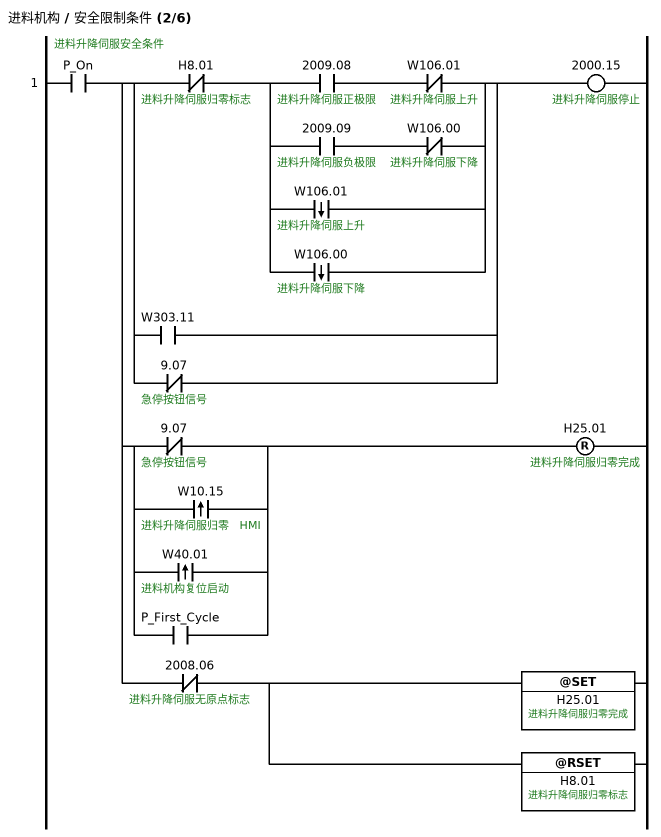
; [picture p72: 进料机构 / 安全限制条件, rungs 1-1]
; rung 1: 进料升降伺服安全条件
LD P_On
OUT TR0
LDNOT H8.01  ; 进料升降伺服归零标志
LD 2009.08  ; 进料升降伺服正极限
ANDNOT W106.01  ; 进料升降伺服上升
LD 2009.09  ; 进料升降伺服负极限
ANDNOT W106.00  ; 进料升降伺服下降
ORLD
%OR W106.01  ; 进料升降伺服上升
%OR W106.00  ; 进料升降伺服下降
ANDLD
OR W303.11
ORNOT 9.07  ; 急停按钮信号
ANDLD
OUT 2000.15  ; 进料升降伺服停止
LD TR0
LDNOT 9.07  ; 急停按钮信号
@OR W10.15  ; 进料升降伺服归零   HMI
@OR W40.01  ; 进料机构复位启动
OR P_First_Cycle
ANDLD
RSET H25.01  ; 进料升降伺服归零完成
LD TR0
ANDNOT 2008.06  ; 进料升降伺服无原点标志
@SET H25.01  ; 进料升降伺服归零完成
@RSET H8.01  ; 进料升降伺服归零标志

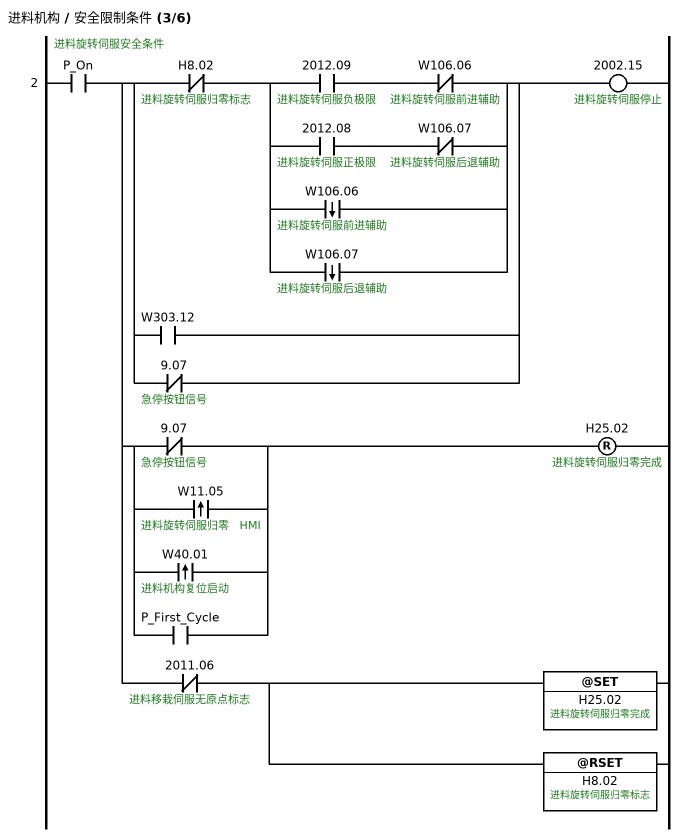
; rung 2: 进料旋转伺服安全条件
LD P_On
OUT TR0
LDNOT H8.02  ; 进料旋转伺服归零标志
LD 2012.09  ; 进料旋转伺服负极限
ANDNOT W106.06  ; 进料旋转伺服前进辅助
LD 2012.08  ; 进料旋转伺服正极限
ANDNOT W106.07  ; 进料旋转伺服后退辅助
ORLD
%OR W106.06  ; 进料旋转伺服前进辅助
%OR W106.07  ; 进料旋转伺服后退辅助
ANDLD
OR W303.12
ORNOT 9.07  ; 急停按钮信号
ANDLD
OUT 2002.15  ; 进料旋转伺服停止
LD TR0
LDNOT 9.07  ; 急停按钮信号
@OR W11.05  ; 进料旋转伺服归零   HMI
@OR W40.01  ; 进料机构复位启动
OR P_First_Cycle
ANDLD
RSET H25.02  ; 进料旋转伺服归零完成
LD TR0
ANDNOT 2011.06  ; 进料移栽伺服无原点标志
@SET H25.02  ; 进料旋转伺服归零完成
@RSET H8.02  ; 进料旋转伺服归零标志

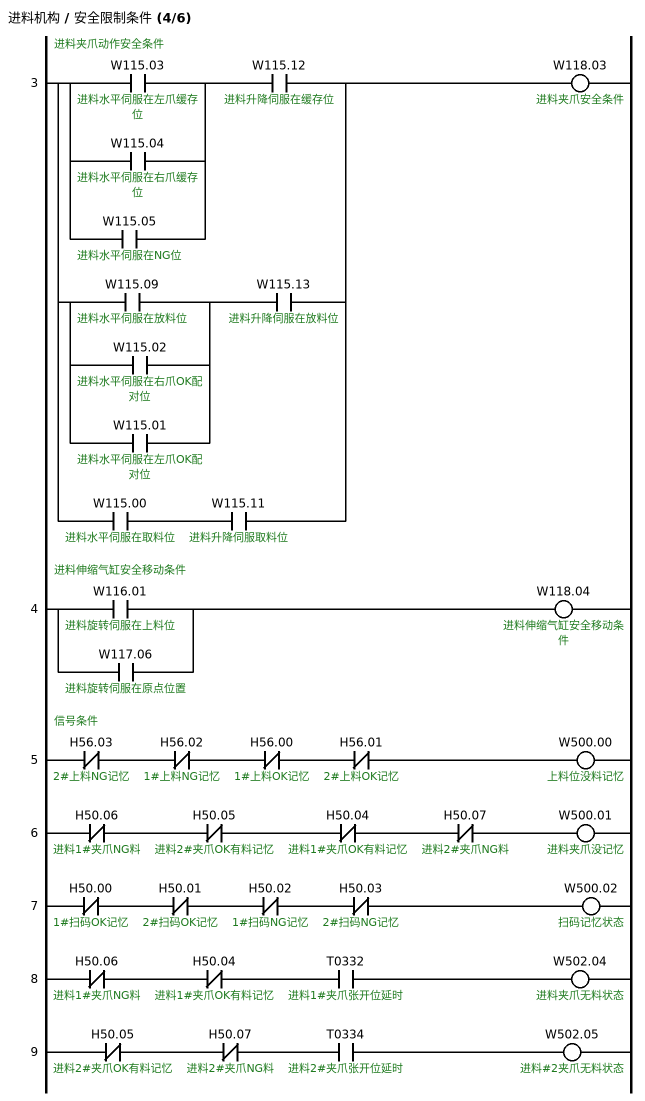
; rung 3: 进料夹爪动作安全条件
LD W115.03  ; 进料水平伺服在左爪缓存位
OR W115.04  ; 进料水平伺服在右爪缓存位
OR W115.05  ; 进料水平伺服在NG位
AND W115.12  ; 进料升降伺服在缓存位
LD W115.09  ; 进料水平伺服在放料位
OR W115.02  ; 进料水平伺服在右爪OK配对位
OR W115.01  ; 进料水平伺服在左爪OK配对位
AND W115.13  ; 进料升降伺服在放料位
ORLD
LD W115.00  ; 进料水平伺服在取料位
AND W115.11  ; 进料升降伺服取料位
ORLD
OUT W118.03  ; 进料夹爪安全条件
; rung 4: 进料伸缩气缸安全移动条件
LD W116.01  ; 进料旋转伺服在上料位
OR W117.06  ; 进料旋转伺服在原点位置
OUT W118.04  ; 进料伸缩气缸安全移动条件
; rung 5: 信号条件
LDNOT H56.03  ; 2#上料NG记忆
ANDNOT H56.02  ; 1#上料NG记忆
ANDNOT H56.00  ; 1#上料OK记忆
ANDNOT H56.01  ; 2#上料OK记忆
OUT W500.00  ; 上料位没料记忆
; rung 6
LDNOT H50.06  ; 进料1#夹爪NG料
ANDNOT H50.05  ; 进料2#夹爪OK有料记忆
ANDNOT H50.04  ; 进料1#夹爪OK有料记忆
ANDNOT H50.07  ; 进料2#夹爪NG料
OUT W500.01  ; 进料夹爪没记忆
; rung 7
LDNOT H50.00  ; 1#扫码OK记忆
ANDNOT H50.01  ; 2#扫码OK记忆
ANDNOT H50.02  ; 1#扫码NG记忆
ANDNOT H50.03  ; 2#扫码NG记忆
OUT W500.02  ; 扫码记忆状态
; rung 8
LDNOT H50.06  ; 进料1#夹爪NG料
ANDNOT H50.04  ; 进料1#夹爪OK有料记忆
AND T0332  ; 进料1#夹爪张开位延时
OUT W502.04  ; 进料夹爪无料状态
; rung 9
LDNOT H50.05  ; 进料2#夹爪OK有料记忆
ANDNOT H50.07  ; 进料2#夹爪NG料
AND T0334  ; 进料2#夹爪张开位延时
OUT W502.05  ; 进料#2夹爪无料状态

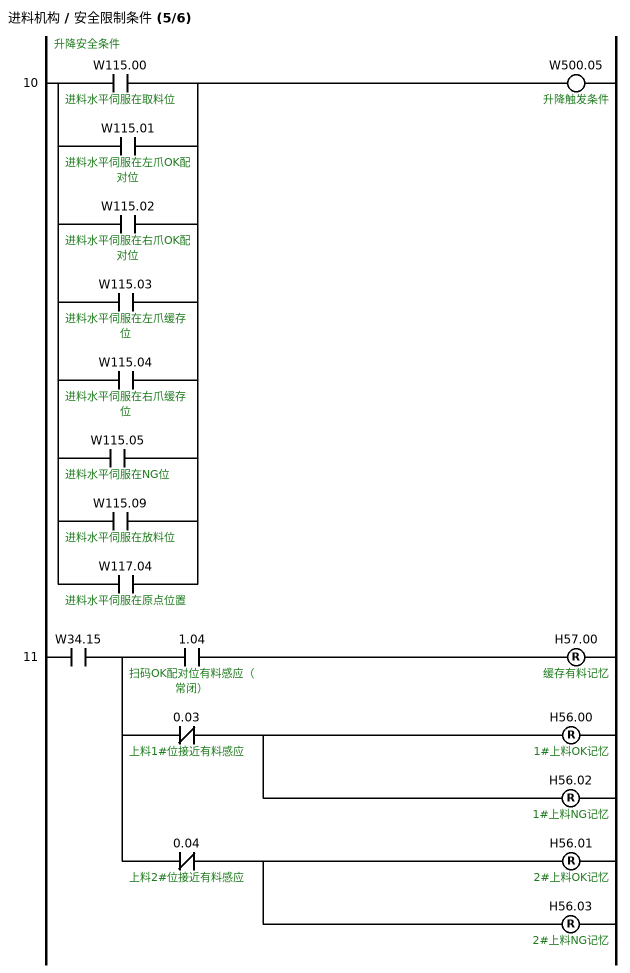
; rung 10: 升降安全条件
LD W115.00  ; 进料水平伺服在取料位
OR W115.01  ; 进料水平伺服在左爪OK配对位
OR W115.02  ; 进料水平伺服在右爪OK配对位
OR W115.03  ; 进料水平伺服在左爪缓存位
OR W115.04  ; 进料水平伺服在右爪缓存位
OR W115.05  ; 进料水平伺服在NG位
OR W115.09  ; 进料水平伺服在放料位
OR W117.04  ; 进料水平伺服在原点位置
OUT W500.05  ; 升降触发条件
; rung 11
LD W34.15
OUT TR0
AND 1.04  ; 扫码OK配对位有料感应（常闭）
RSET H57.00  ; 缓存有料记忆
LD TR0
ANDNOT 0.03  ; 上料1#位接近有料感应
RSET H56.00  ; 1#上料OK记忆
RSET H56.02  ; 1#上料NG记忆
LD TR0
ANDNOT 0.04  ; 上料2#位接近有料感应
RSET H56.01  ; 2#上料OK记忆
RSET H56.03  ; 2#上料NG记忆

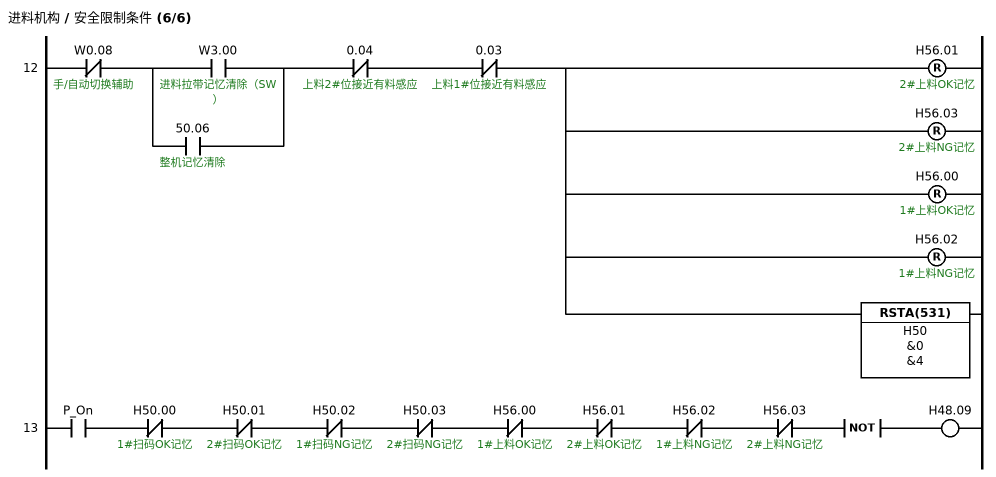
; rung 12
LDNOT W0.08  ; 手/自动切换辅助
LD W3.00  ; 进料拉带记忆清除（SW）
OR 50.06  ; 整机记忆清除
ANDLD
ANDNOT 0.04  ; 上料2#位接近有料感应
ANDNOT 0.03  ; 上料1#位接近有料感应
RSET H56.01  ; 2#上料OK记忆
RSET H56.03  ; 2#上料NG记忆
RSET H56.00  ; 1#上料OK记忆
RSET H56.02  ; 1#上料NG记忆
RSTA(531) H50 &0 &4
; rung 13
LD P_On
ANDNOT H50.00  ; 1#扫码OK记忆
ANDNOT H50.01  ; 2#扫码OK记忆
ANDNOT H50.02  ; 1#扫码NG记忆
ANDNOT H50.03  ; 2#扫码NG记忆
ANDNOT H56.00  ; 1#上料OK记忆
ANDNOT H56.01  ; 2#上料OK记忆
ANDNOT H56.02  ; 1#上料NG记忆
ANDNOT H56.03  ; 2#上料NG记忆
NOT(520)
OUT H48.09

### Section 扫码自动

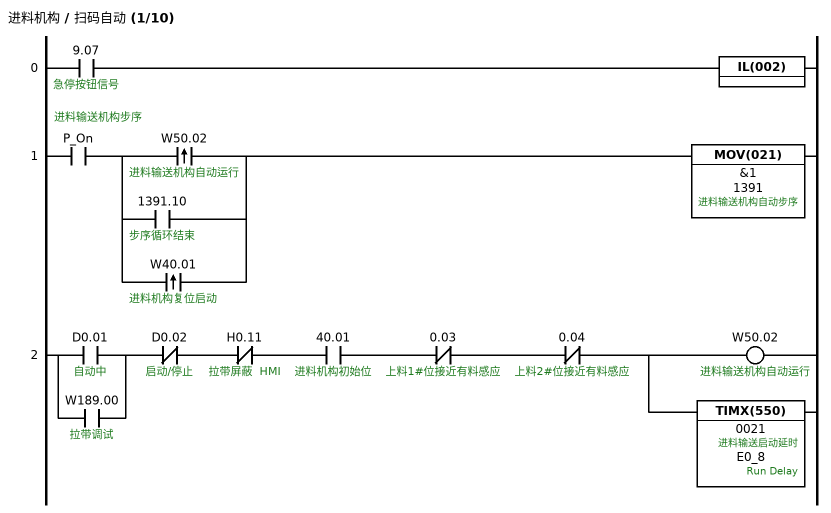
; rung 0
LD 9.07  ; 急停按钮信号
IL(002)
; rung 1: 进料输送机构步序
LD P_On
@LD W50.02  ; 进料输送机构自动运行
OR 1391.10  ; 步序循环结束
@OR W40.01  ; 进料机构复位启动
ANDLD
MOV(021) &1 1391  ; 进料输送机构自动步序
; rung 2
LD D0.01  ; 自动中
OR W189.00  ; 拉带调试
ANDNOT D0.02  ; 启动/停止
ANDNOT H0.11  ; 拉带屏蔽  HMI
AND 40.01  ; 进料机构初始位
ANDNOT 0.03  ; 上料1#位接近有料感应
ANDNOT 0.04  ; 上料2#位接近有料感应
OUT W50.02  ; 进料输送机构自动运行
TIMX(550) 0021 E0_8  ; Run Delay, 进料输送启动延时

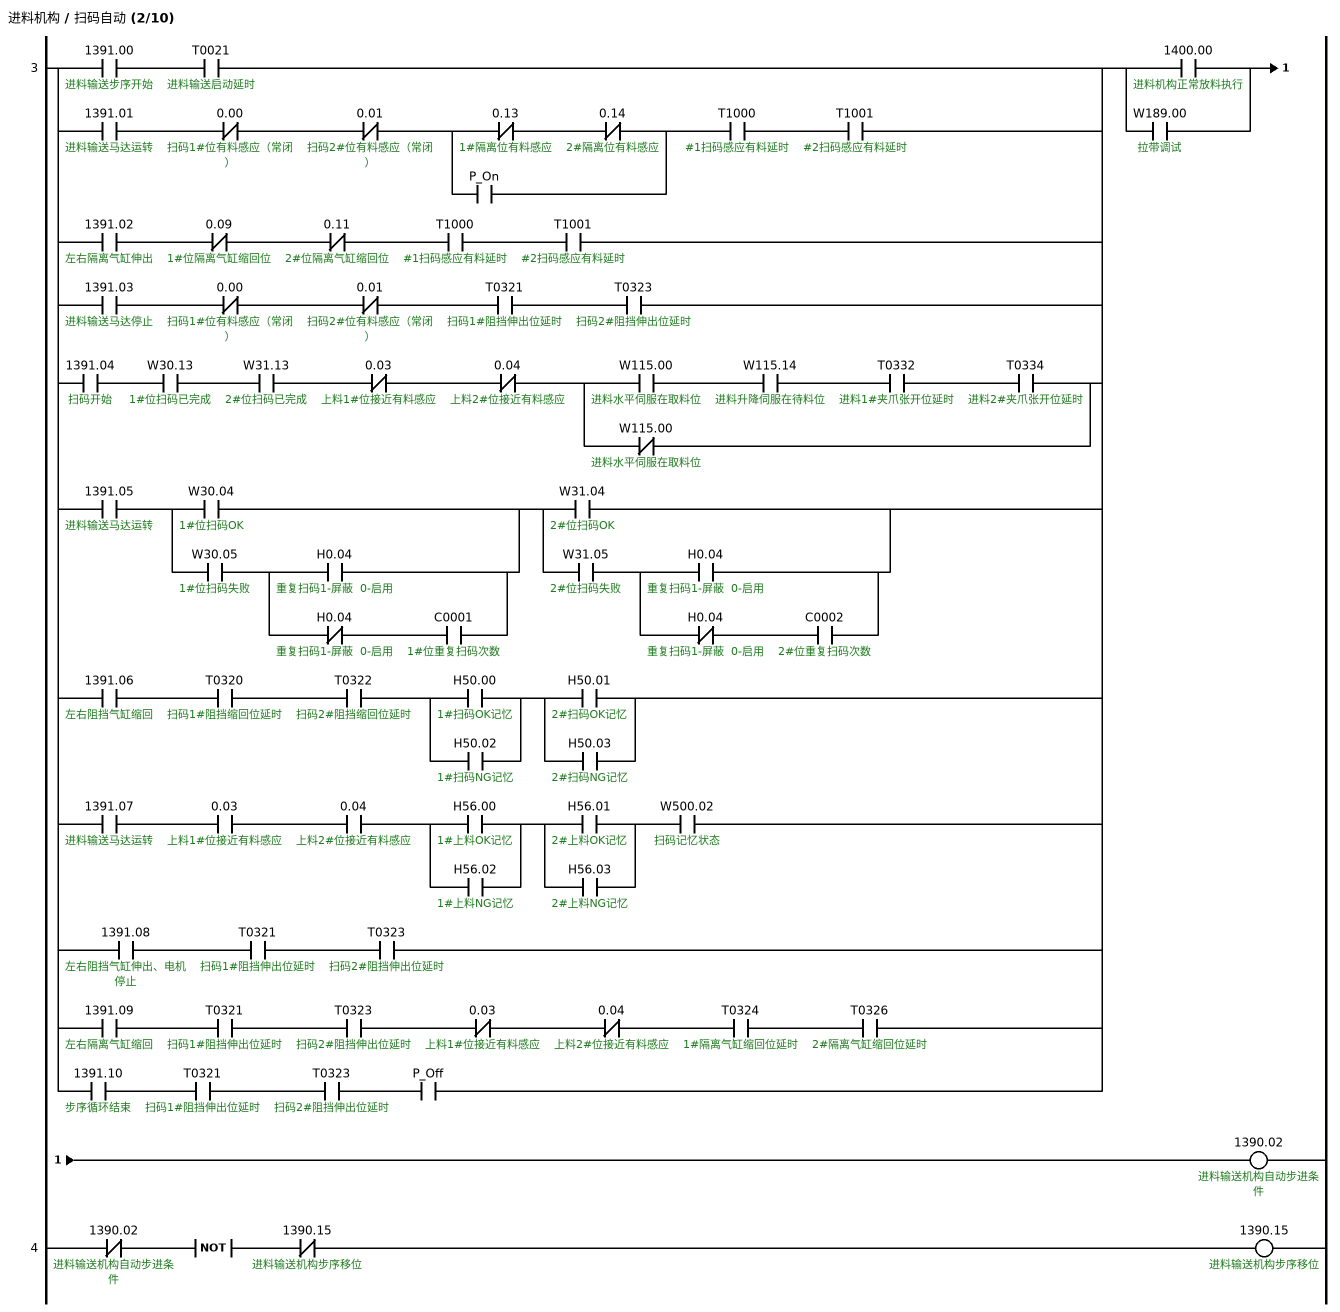
; rung 3
LD 1391.00  ; 进料输送步序开始
AND T0021  ; 进料输送启动延时
LD 1391.01  ; 进料输送马达运转
ANDNOT 0.00  ; 扫码1#位有料感应（常闭）
ANDNOT 0.01  ; 扫码2#位有料感应（常闭）
LDNOT 0.13  ; 1#隔离位有料感应
ANDNOT 0.14  ; 2#隔离位有料感应
OR P_On
ANDLD
AND T1000  ; #1扫码感应有料延时
AND T1001  ; #2扫码感应有料延时
ORLD
LD 1391.02  ; 左右隔离气缸伸出
ANDNOT 0.09  ; 1#位隔离气缸缩回位
ANDNOT 0.11  ; 2#位隔离气缸缩回位
AND T1000  ; #1扫码感应有料延时
AND T1001  ; #2扫码感应有料延时
ORLD
LD 1391.03  ; 进料输送马达停止
ANDNOT 0.00  ; 扫码1#位有料感应（常闭）
ANDNOT 0.01  ; 扫码2#位有料感应（常闭）
AND T0321  ; 扫码1#阻挡伸出位延时
AND T0323  ; 扫码2#阻挡伸出位延时
ORLD
LD 1391.04  ; 扫码开始
AND W30.13  ; 1#位扫码已完成
AND W31.13  ; 2#位扫码已完成
ANDNOT 0.03  ; 上料1#位接近有料感应
ANDNOT 0.04  ; 上料2#位接近有料感应
LD W115.00  ; 进料水平伺服在取料位
AND W115.14  ; 进料升降伺服在待料位
AND T0332  ; 进料1#夹爪张开位延时
AND T0334  ; 进料2#夹爪张开位延时
ORNOT W115.00  ; 进料水平伺服在取料位
ANDLD
ORLD
LD 1391.05  ; 进料输送马达运转
LD W30.04  ; 1#位扫码OK
LD W30.05  ; 1#位扫码失败
LD H0.04  ; 重复扫码1-屏蔽  0-启用
LDNOT H0.04  ; 重复扫码1-屏蔽  0-启用
AND C0001  ; 1#位重复扫码次数
ORLD
ANDLD
ORLD
ANDLD
LD W31.04  ; 2#位扫码OK
LD W31.05  ; 2#位扫码失败
LD H0.04  ; 重复扫码1-屏蔽  0-启用
LDNOT H0.04  ; 重复扫码1-屏蔽  0-启用
AND C0002  ; 2#位重复扫码次数
ORLD
ANDLD
ORLD
ANDLD
ORLD
LD 1391.06  ; 左右阻挡气缸缩回
AND T0320  ; 扫码1#阻挡缩回位延时
AND T0322  ; 扫码2#阻挡缩回位延时
LD H50.00  ; 1#扫码OK记忆
OR H50.02  ; 1#扫码NG记忆
ANDLD
LD H50.01  ; 2#扫码OK记忆
OR H50.03  ; 2#扫码NG记忆
ANDLD
ORLD
LD 1391.07  ; 进料输送马达运转
AND 0.03  ; 上料1#位接近有料感应
AND 0.04  ; 上料2#位接近有料感应
LD H56.00  ; 1#上料OK记忆
OR H56.02  ; 1#上料NG记忆
ANDLD
LD H56.01  ; 2#上料OK记忆
OR H56.03  ; 2#上料NG记忆
ANDLD
AND W500.02  ; 扫码记忆状态
ORLD
LD 1391.08  ; 左右阻挡气缸伸出、电机停止
AND T0321  ; 扫码1#阻挡伸出位延时
AND T0323  ; 扫码2#阻挡伸出位延时
ORLD
LD 1391.09  ; 左右隔离气缸缩回
AND T0321  ; 扫码1#阻挡伸出位延时
AND T0323  ; 扫码2#阻挡伸出位延时
ANDNOT 0.03  ; 上料1#位接近有料感应
ANDNOT 0.04  ; 上料2#位接近有料感应
AND T0324  ; 1#隔离气缸缩回位延时
AND T0326  ; 2#隔离气缸缩回位延时
ORLD
LD 1391.10  ; 步序循环结束
AND T0321  ; 扫码1#阻挡伸出位延时
AND T0323  ; 扫码2#阻挡伸出位延时
AND P_Off
ORLD
LD 1400.00  ; 进料机构正常放料执行
OR W189.00  ; 拉带调试
ANDLD
OUT 1390.02  ; 进料输送机构自动步进条件
; rung 4
LDNOT 1390.02  ; 进料输送机构自动步进条件
NOT(520)
ANDNOT 1390.15  ; 进料输送机构步序移位
OUT 1390.15  ; 进料输送机构步序移位

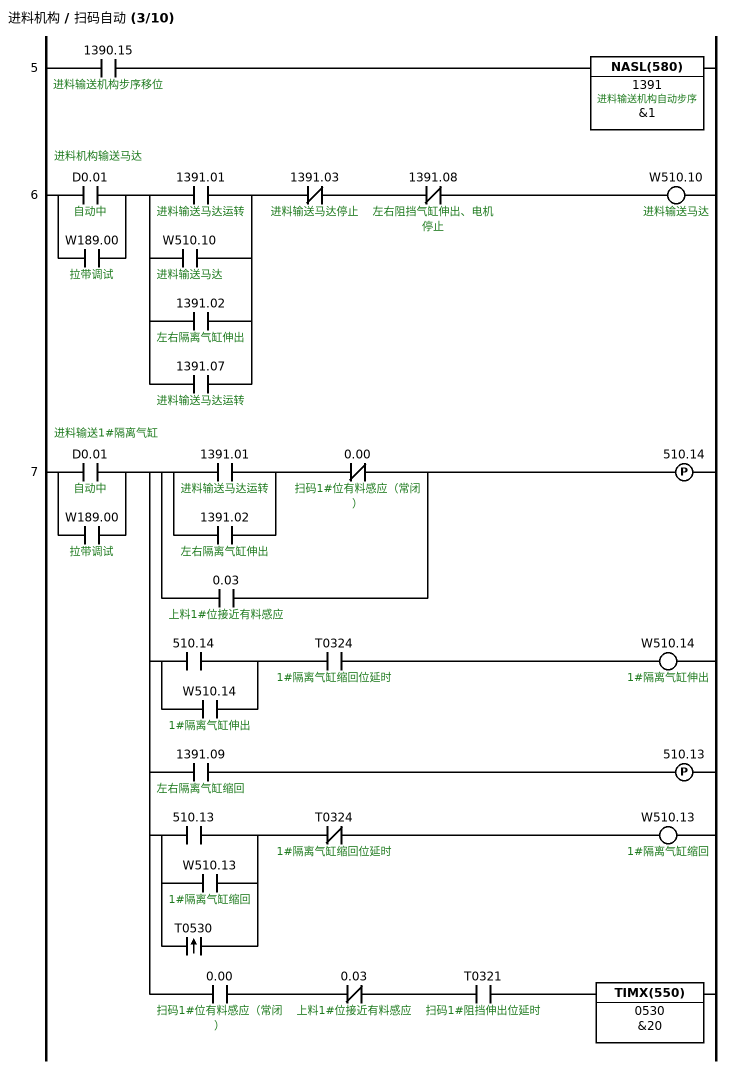
; rung 5
LD 1390.15  ; 进料输送机构步序移位
NASL(580) 1391 &1  ; 进料输送机构自动步序
; rung 6: 进料机构输送马达
LD D0.01  ; 自动中
OR W189.00  ; 拉带调试
LD 1391.01  ; 进料输送马达运转
OR W510.10  ; 进料输送马达
OR 1391.02  ; 左右隔离气缸伸出
OR 1391.07  ; 进料输送马达运转
ANDLD
ANDNOT 1391.03  ; 进料输送马达停止
ANDNOT 1391.08  ; 左右阻挡气缸伸出、电机停止
OUT W510.10  ; 进料输送马达
; rung 7: 进料输送1#隔离气缸
LD D0.01  ; 自动中
OR W189.00  ; 拉带调试
OUT TR0
LD 1391.01  ; 进料输送马达运转
OR 1391.02  ; 左右隔离气缸伸出
ANDNOT 0.00  ; 扫码1#位有料感应（常闭）
OR 0.03  ; 上料1#位接近有料感应
ANDLD
DIFU(013) 510.14
LD TR0
LD 510.14
OR W510.14  ; 1#隔离气缸伸出
ANDLD
AND T0324  ; 1#隔离气缸缩回位延时
OUT W510.14  ; 1#隔离气缸伸出
LD TR0
AND 1391.09  ; 左右隔离气缸缩回
DIFU(013) 510.13
LD TR0
LD 510.13
OR W510.13  ; 1#隔离气缸缩回
@OR T0530
ANDLD
ANDNOT T0324  ; 1#隔离气缸缩回位延时
OUT W510.13  ; 1#隔离气缸缩回
LD TR0
AND 0.00  ; 扫码1#位有料感应（常闭）
ANDNOT 0.03  ; 上料1#位接近有料感应
AND T0321  ; 扫码1#阻挡伸出位延时
TIMX(550) 0530 &20

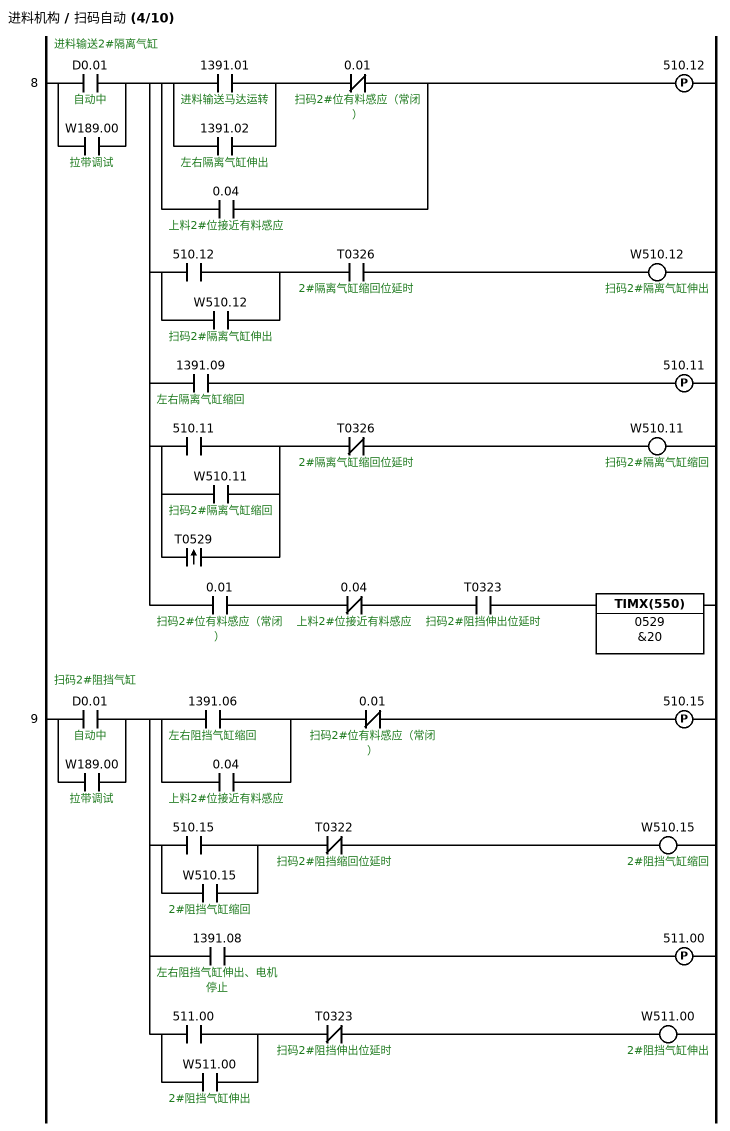
; rung 8: 进料输送2#隔离气缸
LD D0.01  ; 自动中
OR W189.00  ; 拉带调试
OUT TR0
LD 1391.01  ; 进料输送马达运转
OR 1391.02  ; 左右隔离气缸伸出
ANDNOT 0.01  ; 扫码2#位有料感应（常闭）
OR 0.04  ; 上料2#位接近有料感应
ANDLD
DIFU(013) 510.12
LD TR0
LD 510.12
OR W510.12  ; 扫码2#隔离气缸伸出
ANDLD
AND T0326  ; 2#隔离气缸缩回位延时
OUT W510.12  ; 扫码2#隔离气缸伸出
LD TR0
AND 1391.09  ; 左右隔离气缸缩回
DIFU(013) 510.11
LD TR0
LD 510.11
OR W510.11  ; 扫码2#隔离气缸缩回
@OR T0529
ANDLD
ANDNOT T0326  ; 2#隔离气缸缩回位延时
OUT W510.11  ; 扫码2#隔离气缸缩回
LD TR0
AND 0.01  ; 扫码2#位有料感应（常闭）
ANDNOT 0.04  ; 上料2#位接近有料感应
AND T0323  ; 扫码2#阻挡伸出位延时
TIMX(550) 0529 &20
; rung 9: 扫码2#阻挡气缸
LD D0.01  ; 自动中
OR W189.00  ; 拉带调试
OUT TR0
LD 1391.06  ; 左右阻挡气缸缩回
OR 0.04  ; 上料2#位接近有料感应
ANDLD
ANDNOT 0.01  ; 扫码2#位有料感应（常闭）
DIFU(013) 510.15
LD TR0
LD 510.15
OR W510.15  ; 2#阻挡气缸缩回
ANDLD
ANDNOT T0322  ; 扫码2#阻挡缩回位延时
OUT W510.15  ; 2#阻挡气缸缩回
LD TR0
AND 1391.08  ; 左右阻挡气缸伸出、电机停止
DIFU(013) 511.00
LD TR0
LD 511.00
OR W511.00  ; 2#阻挡气缸伸出
ANDLD
ANDNOT T0323  ; 扫码2#阻挡伸出位延时
OUT W511.00  ; 2#阻挡气缸伸出

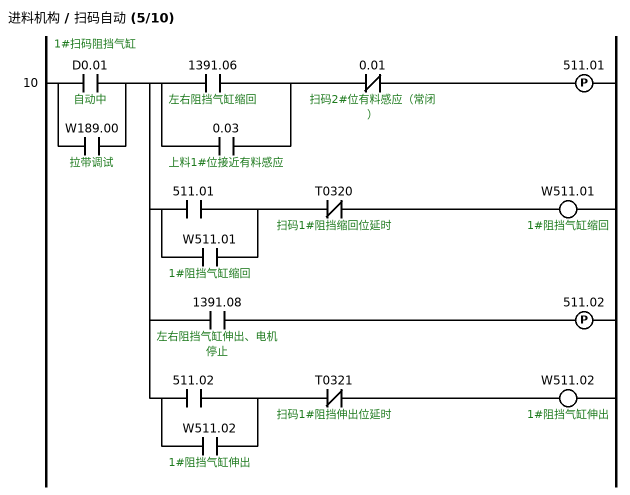
; rung 10: 1#扫码阻挡气缸
LD D0.01  ; 自动中
OR W189.00  ; 拉带调试
OUT TR0
LD 1391.06  ; 左右阻挡气缸缩回
OR 0.03  ; 上料1#位接近有料感应
ANDLD
ANDNOT 0.01  ; 扫码2#位有料感应（常闭）
DIFU(013) 511.01
LD TR0
LD 511.01
OR W511.01  ; 1#阻挡气缸缩回
ANDLD
ANDNOT T0320  ; 扫码1#阻挡缩回位延时
OUT W511.01  ; 1#阻挡气缸缩回
LD TR0
AND 1391.08  ; 左右阻挡气缸伸出、电机停止
DIFU(013) 511.02
LD TR0
LD 511.02
OR W511.02  ; 1#阻挡气缸伸出
ANDLD
ANDNOT T0321  ; 扫码1#阻挡伸出位延时
OUT W511.02  ; 1#阻挡气缸伸出

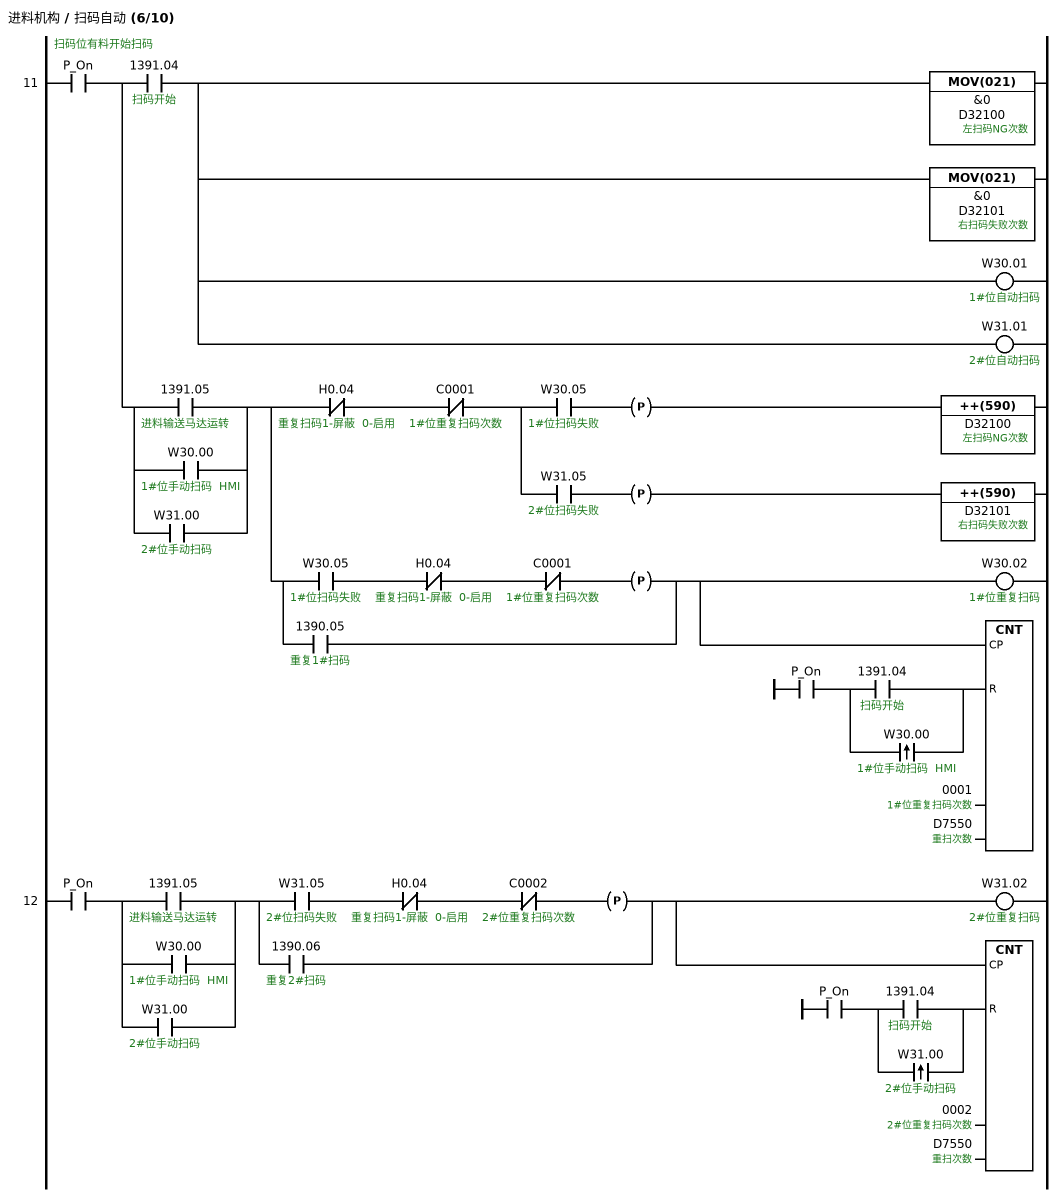
; rung 11: 扫码位有料开始扫码
LD P_On
OUT TR0
AND 1391.04  ; 扫码开始
MOV(021) &0 D32100  ; 左扫码NG次数
MOV(021) &0 D32101  ; 右扫码失败次数
OUT W30.01  ; 1#位自动扫码
OUT W31.01  ; 2#位自动扫码
LD TR0
LD 1391.05  ; 进料输送马达运转
OR W30.00  ; 1#位手动扫码  HMI
OR W31.00  ; 2#位手动扫码
ANDLD
OUT TR0
ANDNOT H0.04  ; 重复扫码1-屏蔽  0-启用
ANDNOT C0001  ; 1#位重复扫码次数
OUT TR1
AND W30.05  ; 1#位扫码失败
UP(521)
++(590) D32100  ; 左扫码NG次数
LD TR1
AND W31.05  ; 2#位扫码失败
UP(521)
++(590) D32101  ; 右扫码失败次数
LD TR0
LD W30.05  ; 1#位扫码失败
ANDNOT H0.04  ; 重复扫码1-屏蔽  0-启用
ANDNOT C0001  ; 1#位重复扫码次数
UP(521)
OR 1390.05  ; 重复1#扫码
ANDLD
OUT W30.02  ; 1#位重复扫码
LD P_On
LD 1391.04  ; 扫码开始
@OR W30.00  ; 1#位手动扫码  HMI
ANDLD
CNT 0001 D7550  ; 重扫次数, 1#位重复扫码次数
; rung 12
LD P_On
LD 1391.05  ; 进料输送马达运转
OR W30.00  ; 1#位手动扫码  HMI
OR W31.00  ; 2#位手动扫码
ANDLD
LD W31.05  ; 2#位扫码失败
ANDNOT H0.04  ; 重复扫码1-屏蔽  0-启用
ANDNOT C0002  ; 2#位重复扫码次数
UP(521)
OR 1390.06  ; 重复2#扫码
ANDLD
OUT W31.02  ; 2#位重复扫码
LD P_On
LD 1391.04  ; 扫码开始
@OR W31.00  ; 2#位手动扫码
ANDLD
CNT 0002 D7550  ; 重扫次数, 2#位重复扫码次数

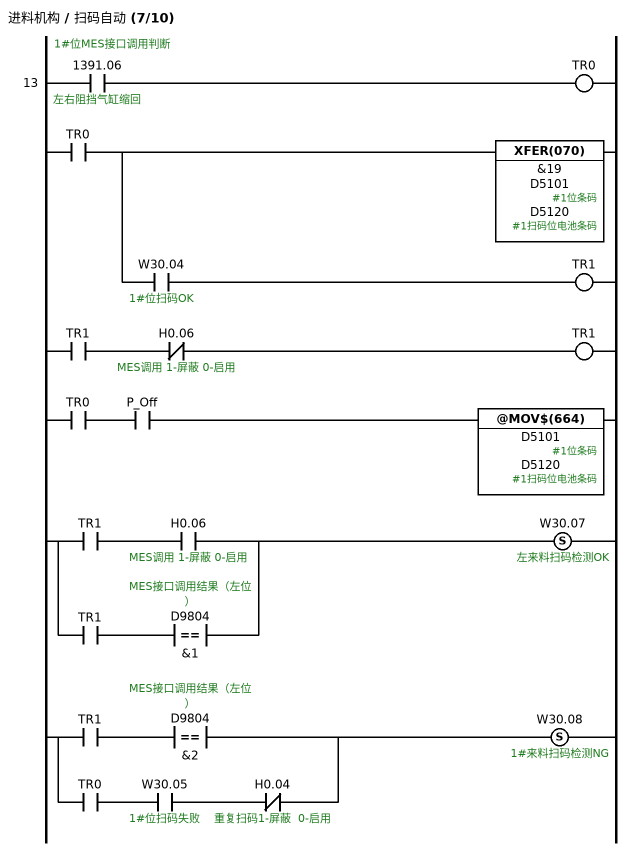
; rung 13: 1#位MES接口调用判断
LD 1391.06  ; 左右阻挡气缸缩回
OUT TR0
AND P_Off
@MOV$(664) D5101 D5120  ; #1位条码, #1扫码位电池条码
LD TR0
XFER(070) &19 D5101 D5120  ; #1位条码, #1扫码位电池条码
AND W30.04  ; 1#位扫码OK
OUT TR1
AND H0.06  ; MES调用 1-屏蔽 0-启用
LD TR1
ANDNOT H0.06  ; MES调用 1-屏蔽 0-启用
OUT TR1
AND=(300) D9804 &1  ; MES接口调用结果（左位）
ORLD
SET W30.07  ; 左来料扫码检测OK
LD TR1
AND=(300) D9804 &2  ; MES接口调用结果（左位）
LD TR0
AND W30.05  ; 1#位扫码失败
ANDNOT H0.04  ; 重复扫码1-屏蔽  0-启用
ORLD
SET W30.08  ; 1#来料扫码检测NG

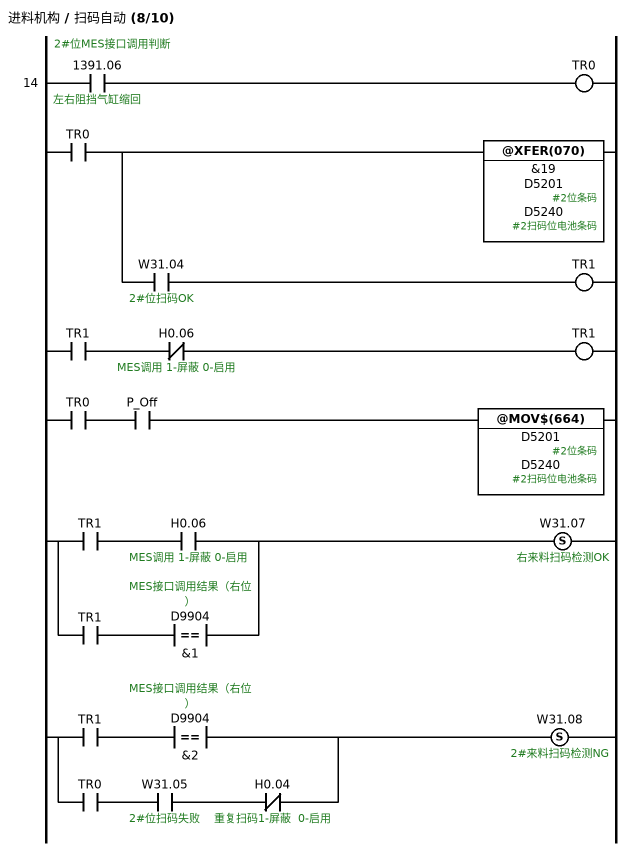
; rung 14: 2#位MES接口调用判断
LD 1391.06  ; 左右阻挡气缸缩回
OUT TR0
AND P_Off
@MOV$(664) D5201 D5240  ; #2位条码, #2扫码位电池条码
LD TR0
@XFER(070) &19 D5201 D5240  ; #2位条码, #2扫码位电池条码
AND W31.04  ; 2#位扫码OK
OUT TR1
AND H0.06  ; MES调用 1-屏蔽 0-启用
LD TR1
ANDNOT H0.06  ; MES调用 1-屏蔽 0-启用
OUT TR1
AND=(300) D9904 &1  ; MES接口调用结果（右位）
ORLD
SET W31.07  ; 右来料扫码检测OK
LD TR1
AND=(300) D9904 &2  ; MES接口调用结果（右位）
LD TR0
AND W31.05  ; 2#位扫码失败
ANDNOT H0.04  ; 重复扫码1-屏蔽  0-启用
ORLD
SET W31.08  ; 2#来料扫码检测NG

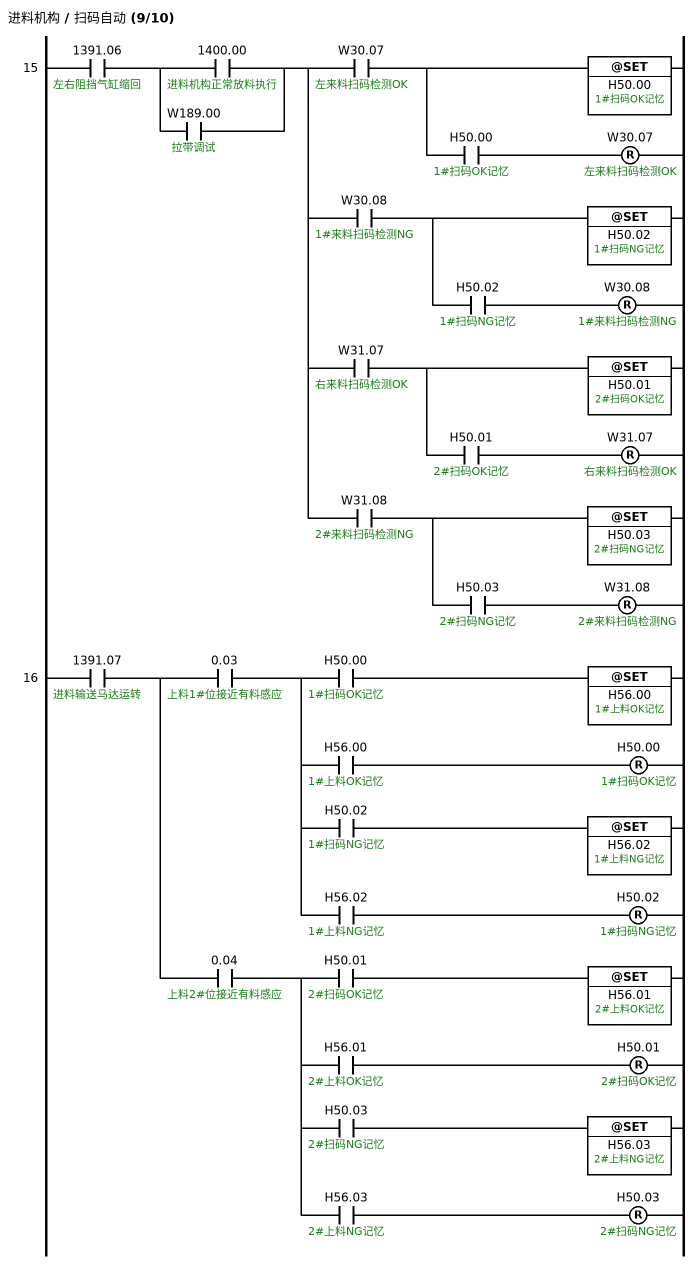
; rung 15
LD 1391.06  ; 左右阻挡气缸缩回
LD 1400.00  ; 进料机构正常放料执行
OR W189.00  ; 拉带调试
ANDLD
OUT TR0
AND W30.07  ; 左来料扫码检测OK
@SET H50.00  ; 1#扫码OK记忆
AND H50.00  ; 1#扫码OK记忆
RSET W30.07  ; 左来料扫码检测OK
LD TR0
AND W30.08  ; 1#来料扫码检测NG
@SET H50.02  ; 1#扫码NG记忆
AND H50.02  ; 1#扫码NG记忆
RSET W30.08  ; 1#来料扫码检测NG
LD TR0
AND W31.07  ; 右来料扫码检测OK
@SET H50.01  ; 2#扫码OK记忆
AND H50.01  ; 2#扫码OK记忆
RSET W31.07  ; 右来料扫码检测OK
LD TR0
AND W31.08  ; 2#来料扫码检测NG
@SET H50.03  ; 2#扫码NG记忆
AND H50.03  ; 2#扫码NG记忆
RSET W31.08  ; 2#来料扫码检测NG
; rung 16
LD 1391.07  ; 进料输送马达运转
OUT TR0
AND 0.03  ; 上料1#位接近有料感应
OUT TR1
AND H50.00  ; 1#扫码OK记忆
@SET H56.00  ; 1#上料OK记忆
LD TR1
AND H56.00  ; 1#上料OK记忆
RSET H50.00  ; 1#扫码OK记忆
LD TR1
AND H50.02  ; 1#扫码NG记忆
@SET H56.02  ; 1#上料NG记忆
LD TR1
AND H56.02  ; 1#上料NG记忆
RSET H50.02  ; 1#扫码NG记忆
LD TR0
AND 0.04  ; 上料2#位接近有料感应
OUT TR0
AND H50.01  ; 2#扫码OK记忆
@SET H56.01  ; 2#上料OK记忆
LD TR0
AND H56.01  ; 2#上料OK记忆
RSET H50.01  ; 2#扫码OK记忆
LD TR0
AND H50.03  ; 2#扫码NG记忆
@SET H56.03  ; 2#上料NG记忆
LD TR0
AND H56.03  ; 2#上料NG记忆
RSET H50.03  ; 2#扫码NG记忆

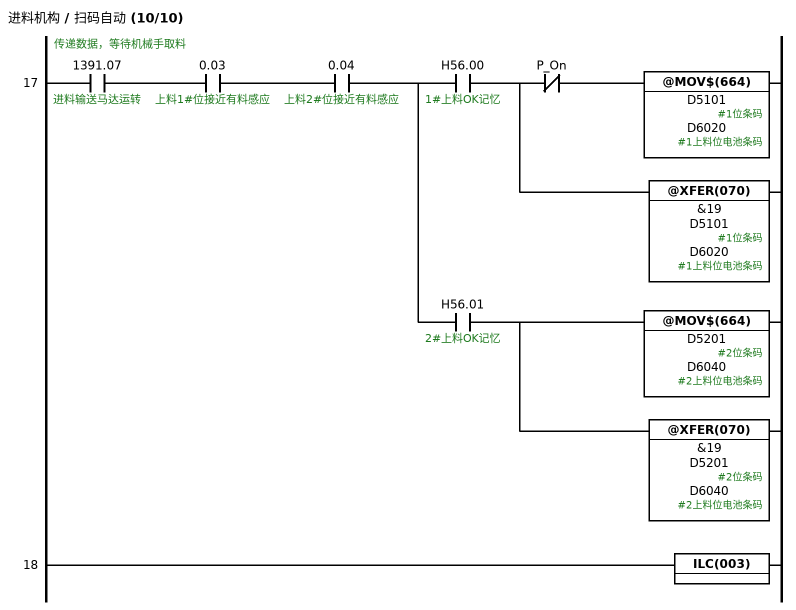
; rung 17: 传递数据，等待机械手取料
LD 1391.07  ; 进料输送马达运转
AND 0.03  ; 上料1#位接近有料感应
AND 0.04  ; 上料2#位接近有料感应
OUT TR0
AND H56.00  ; 1#上料OK记忆
OUT TR1
ANDNOT P_On
@MOV$(664) D5101 D6020  ; #1位条码, #1上料位电池条码
LD TR1
@XFER(070) &19 D5101 D6020  ; #1位条码, #1上料位电池条码
LD TR0
AND H56.01  ; 2#上料OK记忆
@MOV$(664) D5201 D6040  ; #2位条码, #2上料位电池条码
@XFER(070) &19 D5201 D6040  ; #2位条码, #2上料位电池条码
; rung 18
ILC(003)

### Section 进料机构自动

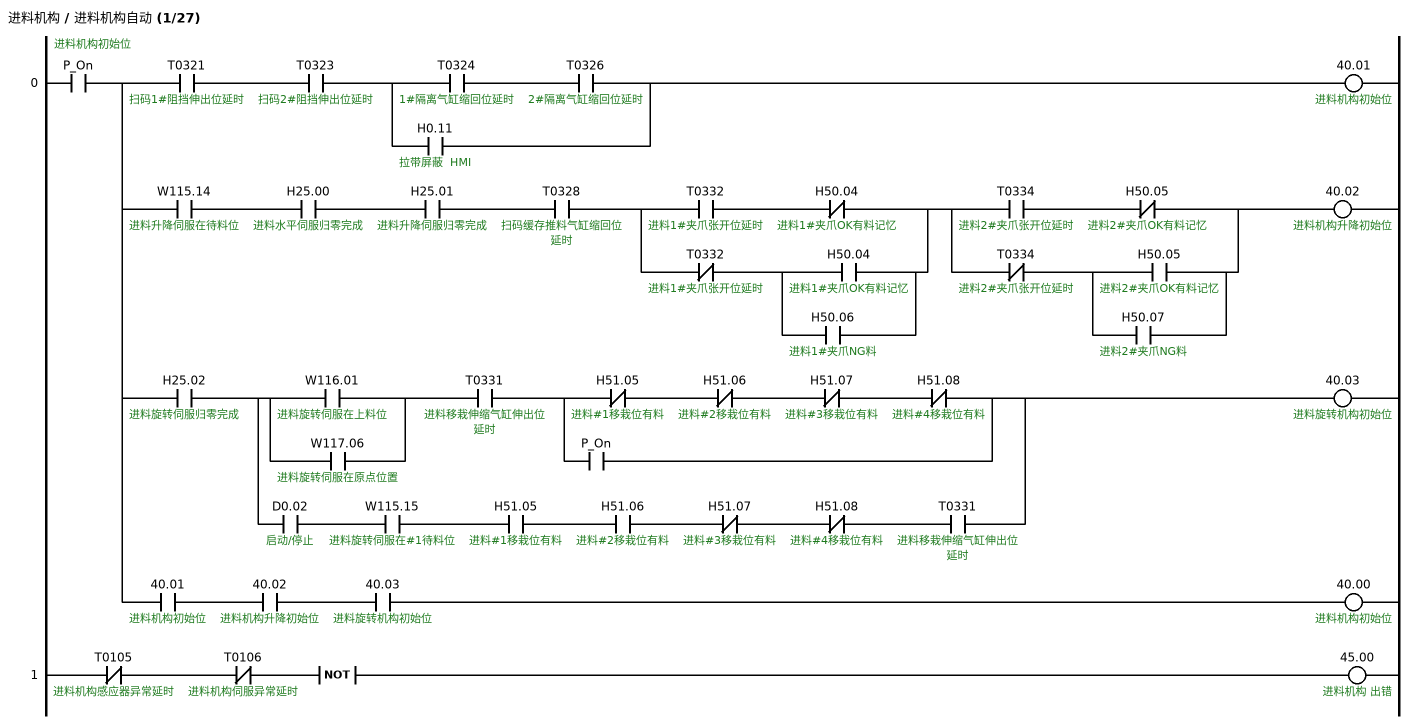
; rung 0: 进料机构初始位
LD P_On
OUT TR0
AND T0321  ; 扫码1#阻挡伸出位延时
AND T0323  ; 扫码2#阻挡伸出位延时
LD T0324  ; 1#隔离气缸缩回位延时
AND T0326  ; 2#隔离气缸缩回位延时
OR H0.11  ; 拉带屏蔽  HMI
ANDLD
OUT 40.01  ; 进料机构初始位
LD TR0
AND W115.14  ; 进料升降伺服在待料位
AND H25.00  ; 进料水平伺服归零完成
AND H25.01  ; 进料升降伺服归零完成
AND T0328  ; 扫码缓存推料气缸缩回位延时
LD T0332  ; 进料1#夹爪张开位延时
ANDNOT H50.04  ; 进料1#夹爪OK有料记忆
LDNOT T0332  ; 进料1#夹爪张开位延时
LD H50.04  ; 进料1#夹爪OK有料记忆
OR H50.06  ; 进料1#夹爪NG料
ANDLD
ORLD
ANDLD
LD T0334  ; 进料2#夹爪张开位延时
ANDNOT H50.05  ; 进料2#夹爪OK有料记忆
LDNOT T0334  ; 进料2#夹爪张开位延时
LD H50.05  ; 进料2#夹爪OK有料记忆
OR H50.07  ; 进料2#夹爪NG料
ANDLD
ORLD
ANDLD
OUT 40.02  ; 进料机构升降初始位
LD TR0
AND H25.02  ; 进料旋转伺服归零完成
LD W116.01  ; 进料旋转伺服在上料位
OR W117.06  ; 进料旋转伺服在原点位置
AND T0331  ; 进料移栽伸缩气缸伸出位延时
LDNOT H51.05  ; 进料#1移栽位有料
ANDNOT H51.06  ; 进料#2移栽位有料
ANDNOT H51.07  ; 进料#3移栽位有料
ANDNOT H51.08  ; 进料#4移栽位有料
OR P_On
ANDLD
LD D0.02  ; 启动/停止
AND W115.15  ; 进料旋转伺服在#1待料位
AND H51.05  ; 进料#1移栽位有料
AND H51.06  ; 进料#2移栽位有料
ANDNOT H51.07  ; 进料#3移栽位有料
ANDNOT H51.08  ; 进料#4移栽位有料
AND T0331  ; 进料移栽伸缩气缸伸出位延时
ORLD
ANDLD
OUT 40.03  ; 进料旋转机构初始位
LD TR0
AND 40.01  ; 进料机构初始位
AND 40.02  ; 进料机构升降初始位
AND 40.03  ; 进料旋转机构初始位
OUT 40.00  ; 进料机构初始位
; rung 1
LDNOT T0105  ; 进料机构感应器异常延时
ANDNOT T0106  ; 进料机构伺服异常延时
NOT(520)
OUT 45.00  ; 进料机构 出错

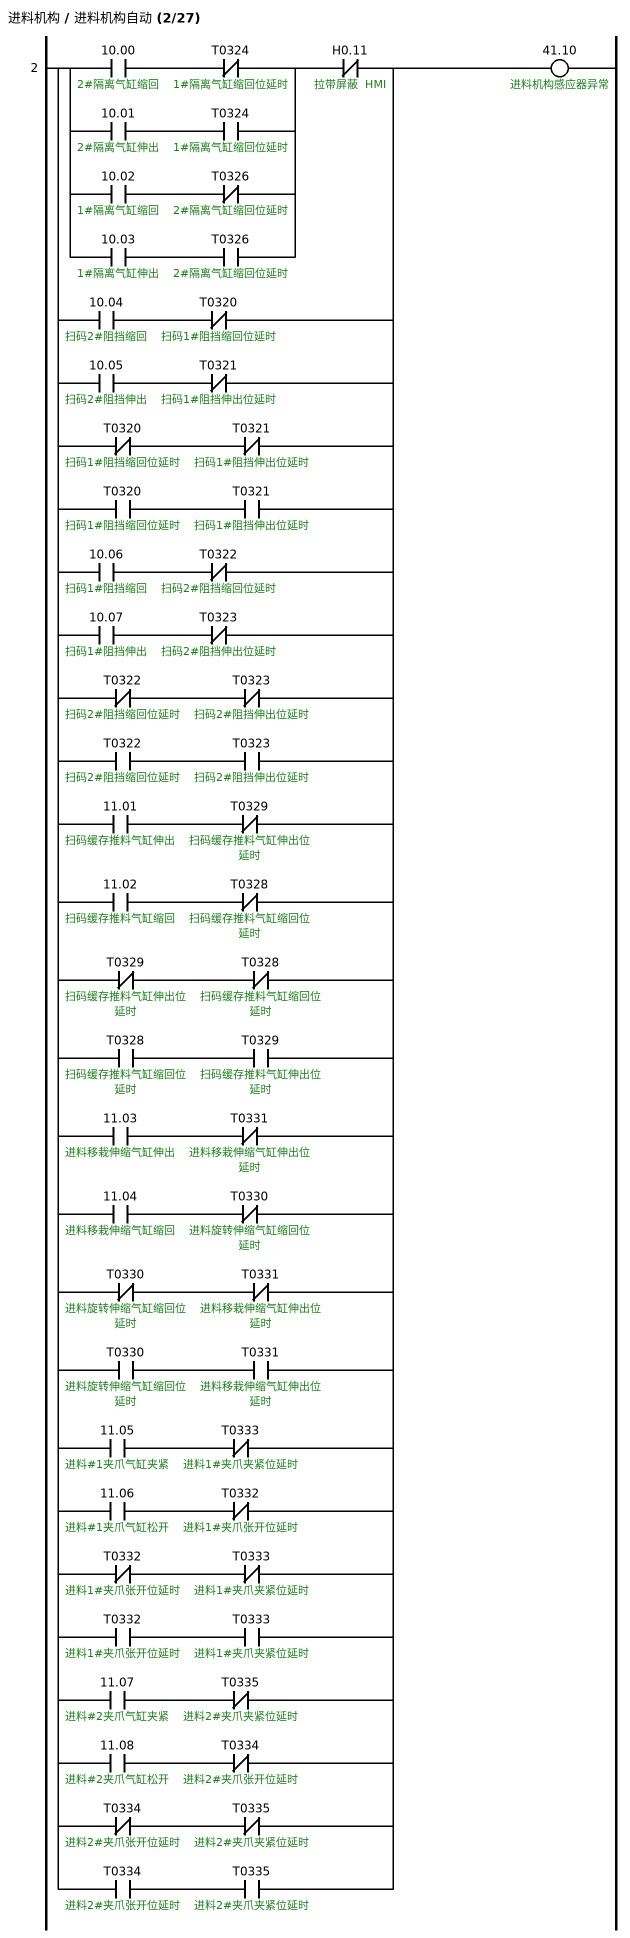
; rung 2
LD 10.00  ; 2#隔离气缸缩回
ANDNOT T0324  ; 1#隔离气缸缩回位延时
LD 10.01  ; 2#隔离气缸伸出
AND T0324  ; 1#隔离气缸缩回位延时
ORLD
LD 10.02  ; 1#隔离气缸缩回
ANDNOT T0326  ; 2#隔离气缸缩回位延时
ORLD
LD 10.03  ; 1#隔离气缸伸出
AND T0326  ; 2#隔离气缸缩回位延时
ORLD
ANDNOT H0.11  ; 拉带屏蔽  HMI
LD 10.04  ; 扫码2#阻挡缩回
ANDNOT T0320  ; 扫码1#阻挡缩回位延时
ORLD
LD 10.05  ; 扫码2#阻挡伸出
ANDNOT T0321  ; 扫码1#阻挡伸出位延时
ORLD
LDNOT T0320  ; 扫码1#阻挡缩回位延时
ANDNOT T0321  ; 扫码1#阻挡伸出位延时
ORLD
LD T0320  ; 扫码1#阻挡缩回位延时
AND T0321  ; 扫码1#阻挡伸出位延时
ORLD
LD 10.06  ; 扫码1#阻挡缩回
ANDNOT T0322  ; 扫码2#阻挡缩回位延时
ORLD
LD 10.07  ; 扫码1#阻挡伸出
ANDNOT T0323  ; 扫码2#阻挡伸出位延时
ORLD
LDNOT T0322  ; 扫码2#阻挡缩回位延时
ANDNOT T0323  ; 扫码2#阻挡伸出位延时
ORLD
LD T0322  ; 扫码2#阻挡缩回位延时
AND T0323  ; 扫码2#阻挡伸出位延时
ORLD
LD 11.01  ; 扫码缓存推料气缸伸出
ANDNOT T0329  ; 扫码缓存推料气缸伸出位延时
ORLD
LD 11.02  ; 扫码缓存推料气缸缩回
ANDNOT T0328  ; 扫码缓存推料气缸缩回位延时
ORLD
LDNOT T0329  ; 扫码缓存推料气缸伸出位延时
ANDNOT T0328  ; 扫码缓存推料气缸缩回位延时
ORLD
LD T0328  ; 扫码缓存推料气缸缩回位延时
AND T0329  ; 扫码缓存推料气缸伸出位延时
ORLD
LD 11.03  ; 进料移栽伸缩气缸伸出
ANDNOT T0331  ; 进料移栽伸缩气缸伸出位延时
ORLD
LD 11.04  ; 进料移栽伸缩气缸缩回
ANDNOT T0330  ; 进料旋转伸缩气缸缩回位延时
ORLD
LDNOT T0330  ; 进料旋转伸缩气缸缩回位延时
ANDNOT T0331  ; 进料移栽伸缩气缸伸出位延时
ORLD
LD T0330  ; 进料旋转伸缩气缸缩回位延时
AND T0331  ; 进料移栽伸缩气缸伸出位延时
ORLD
LD 11.05  ; 进料#1夹爪气缸夹紧
ANDNOT T0333  ; 进料1#夹爪夹紧位延时
ORLD
LD 11.06  ; 进料#1夹爪气缸松开
ANDNOT T0332  ; 进料1#夹爪张开位延时
ORLD
LDNOT T0332  ; 进料1#夹爪张开位延时
ANDNOT T0333  ; 进料1#夹爪夹紧位延时
ORLD
LD T0332  ; 进料1#夹爪张开位延时
AND T0333  ; 进料1#夹爪夹紧位延时
ORLD
LD 11.07  ; 进料#2夹爪气缸夹紧
ANDNOT T0335  ; 进料2#夹爪夹紧位延时
ORLD
LD 11.08  ; 进料#2夹爪气缸松开
ANDNOT T0334  ; 进料2#夹爪张开位延时
ORLD
LDNOT T0334  ; 进料2#夹爪张开位延时
ANDNOT T0335  ; 进料2#夹爪夹紧位延时
ORLD
LD T0334  ; 进料2#夹爪张开位延时
AND T0335  ; 进料2#夹爪夹紧位延时
ORLD
OUT 41.10  ; 进料机构感应器异常

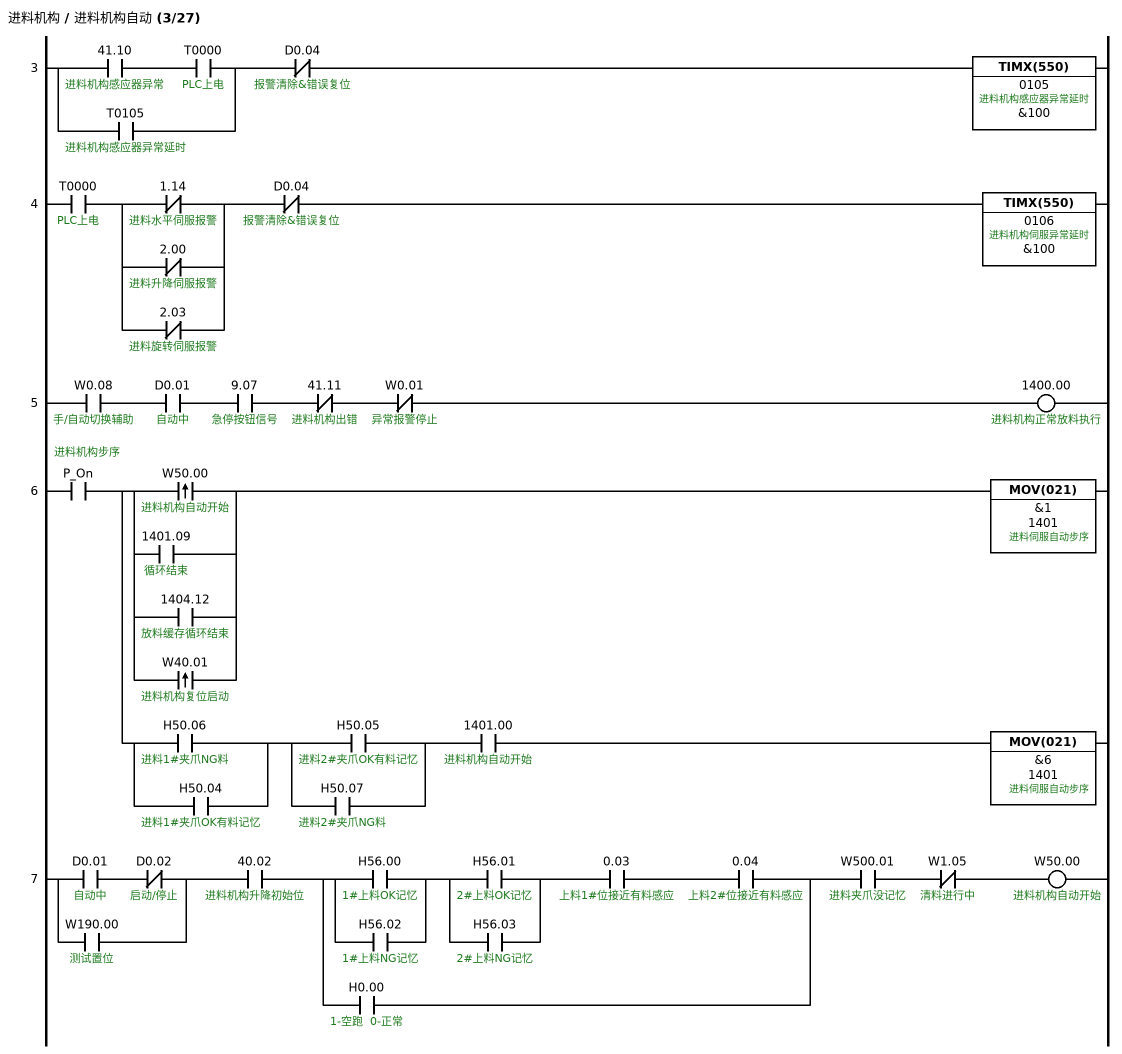
; rung 3
LD 41.10  ; 进料机构感应器异常
AND T0000  ; PLC上电
OR T0105  ; 进料机构感应器异常延时
ANDNOT D0.04  ; 报警清除&错误复位
TIMX(550) 0105 &100  ; 进料机构感应器异常延时
; rung 4
LD T0000  ; PLC上电
LDNOT 1.14  ; 进料水平伺服报警
ORNOT 2.00  ; 进料升降伺服报警
ORNOT 2.03  ; 进料旋转伺服报警
ANDLD
ANDNOT D0.04  ; 报警清除&错误复位
TIMX(550) 0106 &100  ; 进料机构伺服异常延时
; rung 5
LD W0.08  ; 手/自动切换辅助
AND D0.01  ; 自动中
AND 9.07  ; 急停按钮信号
ANDNOT 41.11  ; 进料机构出错
ANDNOT W0.01  ; 异常报警停止
OUT 1400.00  ; 进料机构正常放料执行
; rung 6: 进料机构步序
LD P_On
OUT TR0
@LD W50.00  ; 进料机构自动开始
OR 1401.09  ; 循环结束
OR 1404.12  ; 放料缓存循环结束
@OR W40.01  ; 进料机构复位启动
ANDLD
MOV(021) &1 1401  ; 进料伺服自动步序
LD TR0
LD H50.06  ; 进料1#夹爪NG料
OR H50.04  ; 进料1#夹爪OK有料记忆
ANDLD
LD H50.05  ; 进料2#夹爪OK有料记忆
OR H50.07  ; 进料2#夹爪NG料
ANDLD
AND 1401.00  ; 进料机构自动开始
MOV(021) &6 1401  ; 进料伺服自动步序
; rung 7
LD D0.01  ; 自动中
ANDNOT D0.02  ; 启动/停止
OR W190.00  ; 测试置位
AND 40.02  ; 进料机构升降初始位
LD H56.00  ; 1#上料OK记忆
OR H56.02  ; 1#上料NG记忆
LD H56.01  ; 2#上料OK记忆
OR H56.03  ; 2#上料NG记忆
ANDLD
AND 0.03  ; 上料1#位接近有料感应
AND 0.04  ; 上料2#位接近有料感应
OR H0.00  ; 1-空跑  0-正常
ANDLD
AND W500.01  ; 进料夹爪没记忆
ANDNOT W1.05  ; 清料进行中
OUT W50.00  ; 进料机构自动开始

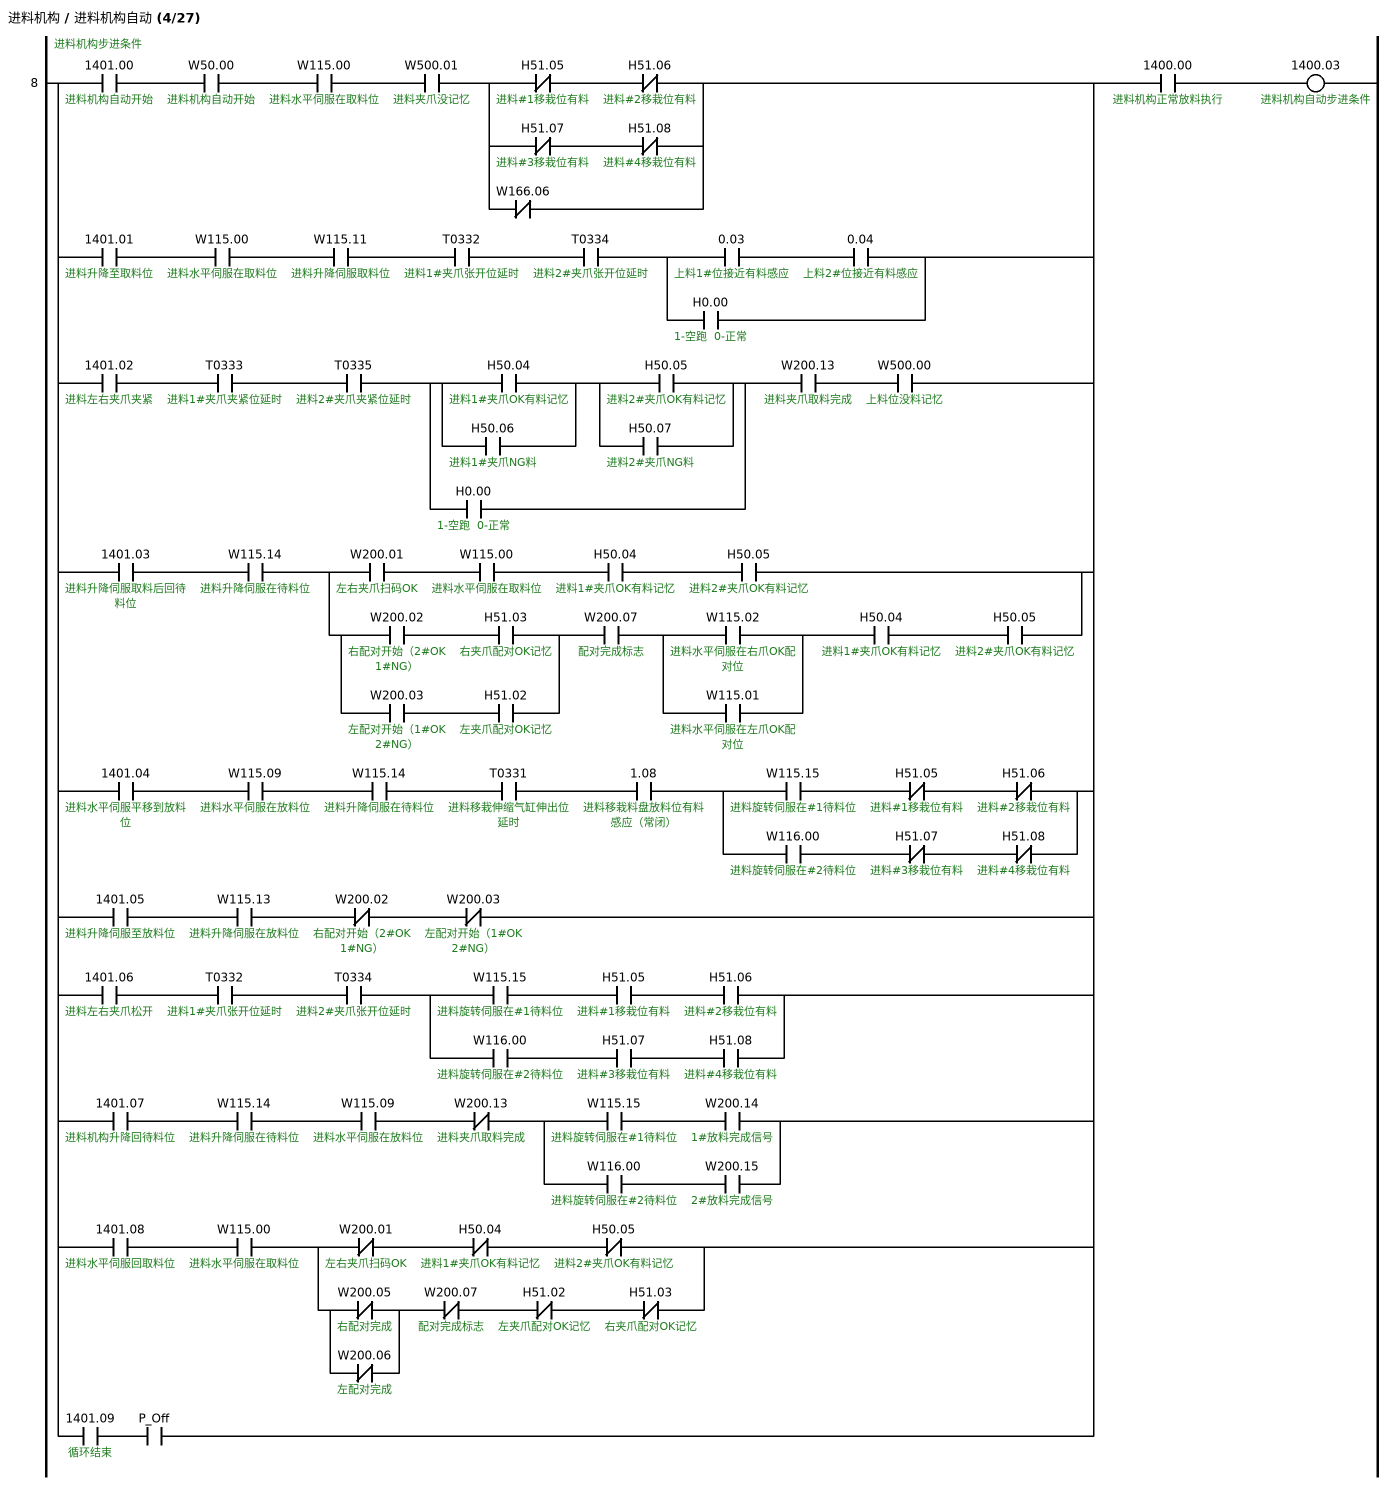
; rung 8: 进料机构步进条件
LD 1401.00  ; 进料机构自动开始
AND W50.00  ; 进料机构自动开始
AND W115.00  ; 进料水平伺服在取料位
AND W500.01  ; 进料夹爪没记忆
LDNOT H51.05  ; 进料#1移栽位有料
ANDNOT H51.06  ; 进料#2移栽位有料
LDNOT H51.07  ; 进料#3移栽位有料
ANDNOT H51.08  ; 进料#4移栽位有料
ORLD
ORNOT W166.06
ANDLD
LD 1401.01  ; 进料升降至取料位
AND W115.00  ; 进料水平伺服在取料位
AND W115.11  ; 进料升降伺服取料位
AND T0332  ; 进料1#夹爪张开位延时
AND T0334  ; 进料2#夹爪张开位延时
LD 0.03  ; 上料1#位接近有料感应
AND 0.04  ; 上料2#位接近有料感应
OR H0.00  ; 1-空跑  0-正常
ANDLD
ORLD
LD 1401.02  ; 进料左右夹爪夹紧
AND T0333  ; 进料1#夹爪夹紧位延时
AND T0335  ; 进料2#夹爪夹紧位延时
LD H50.04  ; 进料1#夹爪OK有料记忆
OR H50.06  ; 进料1#夹爪NG料
LD H50.05  ; 进料2#夹爪OK有料记忆
OR H50.07  ; 进料2#夹爪NG料
ANDLD
OR H0.00  ; 1-空跑  0-正常
ANDLD
AND W200.13  ; 进料夹爪取料完成
AND W500.00  ; 上料位没料记忆
ORLD
LD 1401.03  ; 进料升降伺服取料后回待料位
AND W115.14  ; 进料升降伺服在待料位
LD W200.01  ; 左右夹爪扫码OK
AND W115.00  ; 进料水平伺服在取料位
AND H50.04  ; 进料1#夹爪OK有料记忆
AND H50.05  ; 进料2#夹爪OK有料记忆
LD W200.02  ; 右配对开始（2#OK 1#NG）
AND H51.03  ; 右夹爪配对OK记忆
LD W200.03  ; 左配对开始（1#OK 2#NG）
AND H51.02  ; 左夹爪配对OK记忆
ORLD
AND W200.07  ; 配对完成标志
LD W115.02  ; 进料水平伺服在右爪OK配对位
OR W115.01  ; 进料水平伺服在左爪OK配对位
ANDLD
AND H50.04  ; 进料1#夹爪OK有料记忆
AND H50.05  ; 进料2#夹爪OK有料记忆
ORLD
ANDLD
ORLD
LD 1401.04  ; 进料水平伺服平移到放料位
AND W115.09  ; 进料水平伺服在放料位
AND W115.14  ; 进料升降伺服在待料位
AND T0331  ; 进料移栽伸缩气缸伸出位延时
AND 1.08  ; 进料移栽料盘放料位有料感应（常闭）
LD W115.15  ; 进料旋转伺服在#1待料位
ANDNOT H51.05  ; 进料#1移栽位有料
ANDNOT H51.06  ; 进料#2移栽位有料
LD W116.00  ; 进料旋转伺服在#2待料位
ANDNOT H51.07  ; 进料#3移栽位有料
ANDNOT H51.08  ; 进料#4移栽位有料
ORLD
ANDLD
ORLD
LD 1401.05  ; 进料升降伺服至放料位
AND W115.13  ; 进料升降伺服在放料位
ANDNOT W200.02  ; 右配对开始（2#OK 1#NG）
ANDNOT W200.03  ; 左配对开始（1#OK 2#NG）
ORLD
LD 1401.06  ; 进料左右夹爪松开
AND T0332  ; 进料1#夹爪张开位延时
AND T0334  ; 进料2#夹爪张开位延时
LD W115.15  ; 进料旋转伺服在#1待料位
AND H51.05  ; 进料#1移栽位有料
AND H51.06  ; 进料#2移栽位有料
LD W116.00  ; 进料旋转伺服在#2待料位
AND H51.07  ; 进料#3移栽位有料
AND H51.08  ; 进料#4移栽位有料
ORLD
ANDLD
ORLD
LD 1401.07  ; 进料机构升降回待料位
AND W115.14  ; 进料升降伺服在待料位
AND W115.09  ; 进料水平伺服在放料位
ANDNOT W200.13  ; 进料夹爪取料完成
LD W115.15  ; 进料旋转伺服在#1待料位
AND W200.14  ; 1#放料完成信号
LD W116.00  ; 进料旋转伺服在#2待料位
AND W200.15  ; 2#放料完成信号
ORLD
ANDLD
ORLD
LD 1401.08  ; 进料水平伺服回取料位
AND W115.00  ; 进料水平伺服在取料位
LDNOT W200.01  ; 左右夹爪扫码OK
ANDNOT H50.04  ; 进料1#夹爪OK有料记忆
ANDNOT H50.05  ; 进料2#夹爪OK有料记忆
LDNOT W200.05  ; 右配对完成
ORNOT W200.06  ; 左配对完成
ANDNOT W200.07  ; 配对完成标志
ANDNOT H51.02  ; 左夹爪配对OK记忆
ANDNOT H51.03  ; 右夹爪配对OK记忆
ORLD
ANDLD
ORLD
LD 1401.09  ; 循环结束
AND P_Off
ORLD
AND 1400.00  ; 进料机构正常放料执行
OUT 1400.03  ; 进料机构自动步进条件

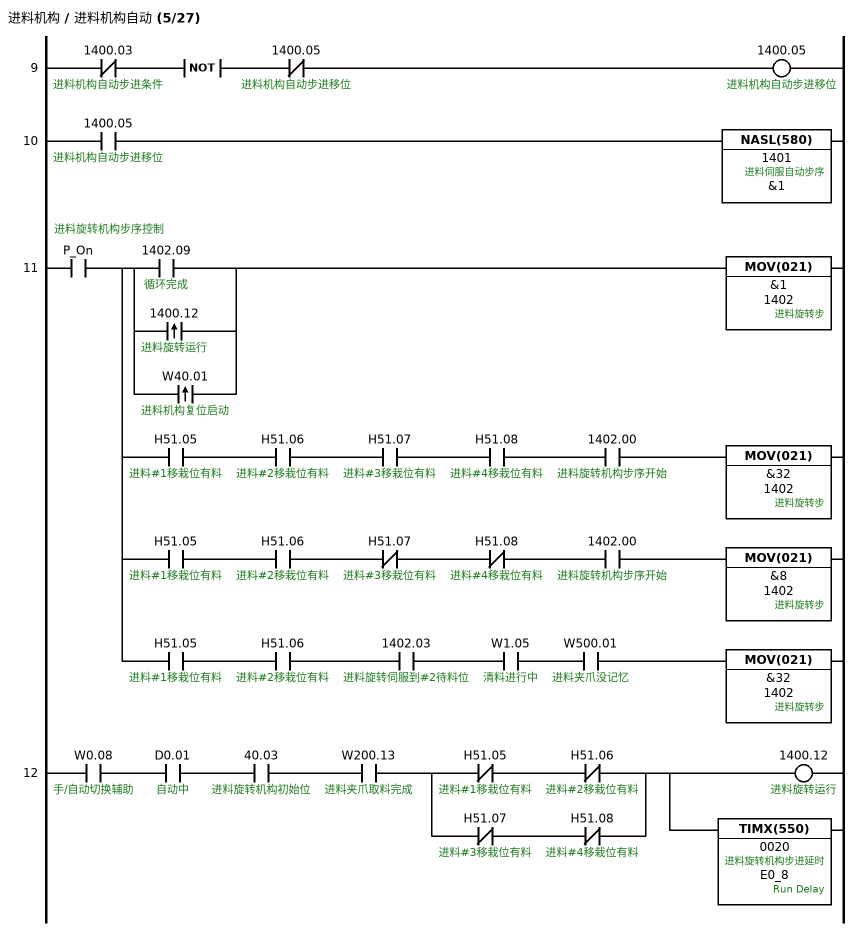
; rung 9
LDNOT 1400.03  ; 进料机构自动步进条件
NOT(520)
ANDNOT 1400.05  ; 进料机构自动步进移位
OUT 1400.05  ; 进料机构自动步进移位
; rung 10
LD 1400.05  ; 进料机构自动步进移位
NASL(580) 1401 &1  ; 进料伺服自动步序
; rung 11: 进料旋转机构步序控制
LD P_On
OUT TR0
LD 1402.09  ; 循环完成
@OR 1400.12  ; 进料旋转运行
@OR W40.01  ; 进料机构复位启动
ANDLD
MOV(021) &1 1402  ; 进料旋转步
LD TR0
AND H51.05  ; 进料#1移栽位有料
AND H51.06  ; 进料#2移栽位有料
AND H51.07  ; 进料#3移栽位有料
AND H51.08  ; 进料#4移栽位有料
AND 1402.00  ; 进料旋转机构步序开始
MOV(021) &32 1402  ; 进料旋转步
LD TR0
AND H51.05  ; 进料#1移栽位有料
AND H51.06  ; 进料#2移栽位有料
ANDNOT H51.07  ; 进料#3移栽位有料
ANDNOT H51.08  ; 进料#4移栽位有料
AND 1402.00  ; 进料旋转机构步序开始
MOV(021) &8 1402  ; 进料旋转步
LD TR0
AND H51.05  ; 进料#1移栽位有料
AND H51.06  ; 进料#2移栽位有料
AND 1402.03  ; 进料旋转伺服到#2待料位
AND W1.05  ; 清料进行中
AND W500.01  ; 进料夹爪没记忆
MOV(021) &32 1402  ; 进料旋转步
; rung 12
LD W0.08  ; 手/自动切换辅助
AND D0.01  ; 自动中
AND 40.03  ; 进料旋转机构初始位
AND W200.13  ; 进料夹爪取料完成
LDNOT H51.05  ; 进料#1移栽位有料
ANDNOT H51.06  ; 进料#2移栽位有料
LDNOT H51.07  ; 进料#3移栽位有料
ANDNOT H51.08  ; 进料#4移栽位有料
ORLD
ANDLD
OUT 1400.12  ; 进料旋转运行
TIMX(550) 0020 E0_8  ; Run Delay, 进料旋转机构步进延时

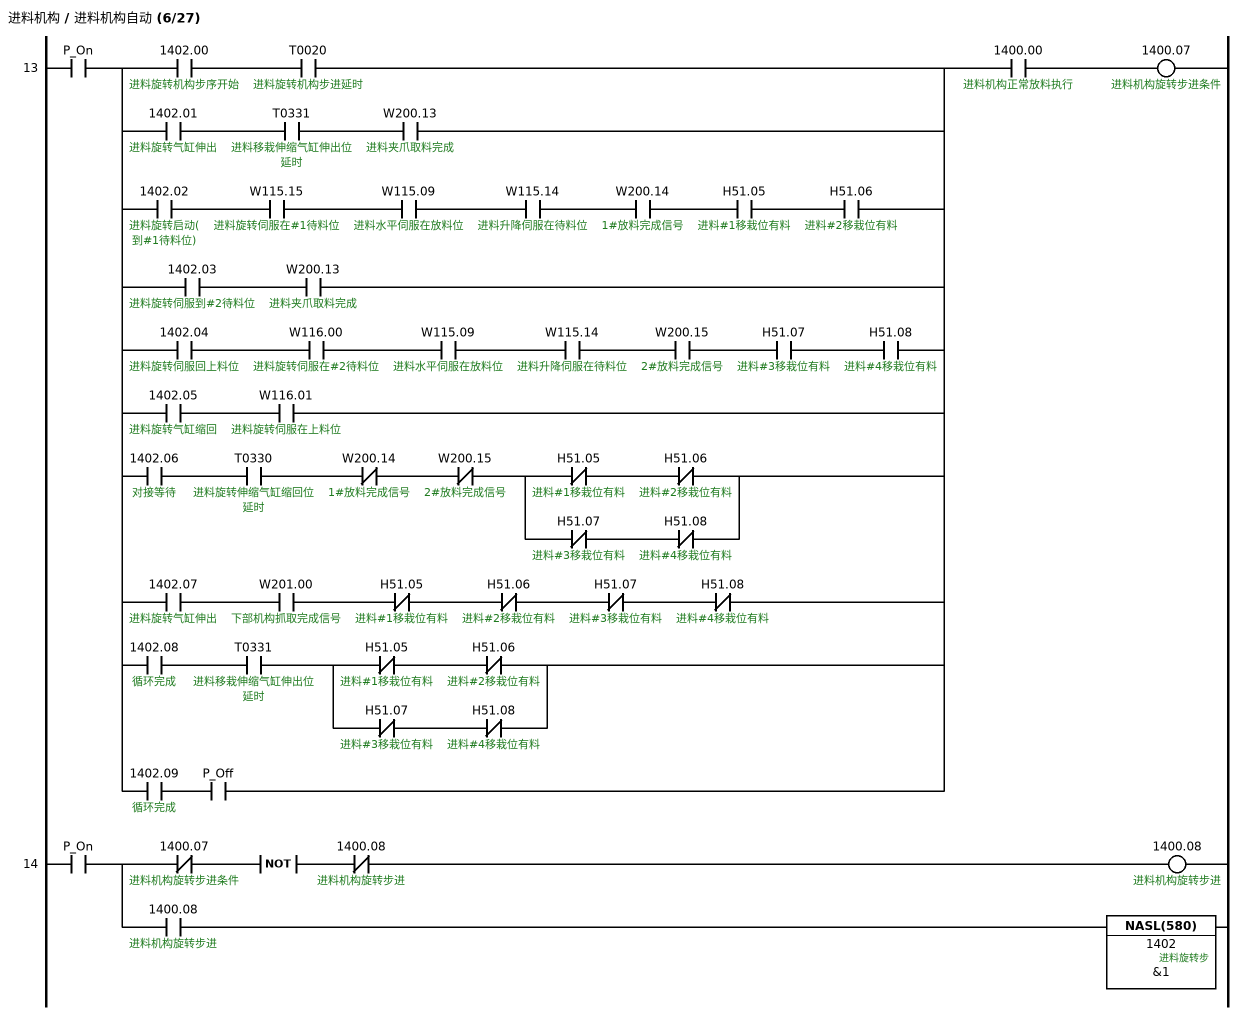
; rung 13
LD P_On
LD 1402.00  ; 进料旋转机构步序开始
AND T0020  ; 进料旋转机构步进延时
LD 1402.01  ; 进料旋转气缸伸出
AND T0331  ; 进料移栽伸缩气缸伸出位延时
AND W200.13  ; 进料夹爪取料完成
ORLD
LD 1402.02  ; 进料旋转启动(到#1待料位)
AND W115.15  ; 进料旋转伺服在#1待料位
AND W115.09  ; 进料水平伺服在放料位
AND W115.14  ; 进料升降伺服在待料位
AND W200.14  ; 1#放料完成信号
AND H51.05  ; 进料#1移栽位有料
AND H51.06  ; 进料#2移栽位有料
ORLD
LD 1402.03  ; 进料旋转伺服到#2待料位
AND W200.13  ; 进料夹爪取料完成
ORLD
LD 1402.04  ; 进料旋转伺服回上料位
AND W116.00  ; 进料旋转伺服在#2待料位
AND W115.09  ; 进料水平伺服在放料位
AND W115.14  ; 进料升降伺服在待料位
AND W200.15  ; 2#放料完成信号
AND H51.07  ; 进料#3移栽位有料
AND H51.08  ; 进料#4移栽位有料
ORLD
LD 1402.05  ; 进料旋转气缸缩回
AND W116.01  ; 进料旋转伺服在上料位
ORLD
LD 1402.06  ; 对接等待
AND T0330  ; 进料旋转伸缩气缸缩回位延时
ANDNOT W200.14  ; 1#放料完成信号
ANDNOT W200.15  ; 2#放料完成信号
LDNOT H51.05  ; 进料#1移栽位有料
ANDNOT H51.06  ; 进料#2移栽位有料
LDNOT H51.07  ; 进料#3移栽位有料
ANDNOT H51.08  ; 进料#4移栽位有料
ORLD
ANDLD
ORLD
LD 1402.07  ; 进料旋转气缸伸出
AND W201.00  ; 下部机构抓取完成信号
ANDNOT H51.05  ; 进料#1移栽位有料
ANDNOT H51.06  ; 进料#2移栽位有料
ANDNOT H51.07  ; 进料#3移栽位有料
ANDNOT H51.08  ; 进料#4移栽位有料
ORLD
LD 1402.08  ; 循环完成
AND T0331  ; 进料移栽伸缩气缸伸出位延时
LDNOT H51.05  ; 进料#1移栽位有料
ANDNOT H51.06  ; 进料#2移栽位有料
LDNOT H51.07  ; 进料#3移栽位有料
ANDNOT H51.08  ; 进料#4移栽位有料
ORLD
ANDLD
ORLD
LD 1402.09  ; 循环完成
AND P_Off
ORLD
ANDLD
AND 1400.00  ; 进料机构正常放料执行
OUT 1400.07  ; 进料机构旋转步进条件
; rung 14
LD P_On
OUT TR0
ANDNOT 1400.07  ; 进料机构旋转步进条件
NOT(520)
ANDNOT 1400.08  ; 进料机构旋转步进
OUT 1400.08  ; 进料机构旋转步进
LD TR0
AND 1400.08  ; 进料机构旋转步进
NASL(580) 1402 &1  ; 进料旋转步

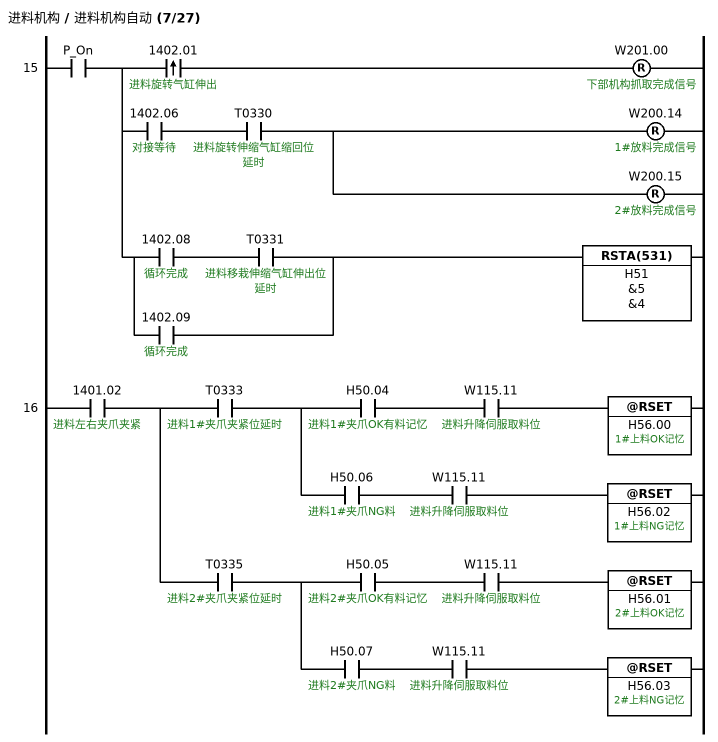
; rung 15
LD P_On
OUT TR0
@AND 1402.01  ; 进料旋转气缸伸出
RSET W201.00  ; 下部机构抓取完成信号
LD TR0
AND 1402.06  ; 对接等待
AND T0330  ; 进料旋转伸缩气缸缩回位延时
RSET W200.14  ; 1#放料完成信号
RSET W200.15  ; 2#放料完成信号
LD TR0
LD 1402.08  ; 循环完成
AND T0331  ; 进料移栽伸缩气缸伸出位延时
OR 1402.09  ; 循环完成
ANDLD
RSTA(531) H51 &5 &4
; rung 16
LD 1401.02  ; 进料左右夹爪夹紧
OUT TR0
AND T0333  ; 进料1#夹爪夹紧位延时
OUT TR1
AND H50.04  ; 进料1#夹爪OK有料记忆
AND W115.11  ; 进料升降伺服取料位
@RSET H56.00  ; 1#上料OK记忆
LD TR1
AND H50.06  ; 进料1#夹爪NG料
AND W115.11  ; 进料升降伺服取料位
@RSET H56.02  ; 1#上料NG记忆
LD TR0
AND T0335  ; 进料2#夹爪夹紧位延时
OUT TR0
AND H50.05  ; 进料2#夹爪OK有料记忆
AND W115.11  ; 进料升降伺服取料位
@RSET H56.01  ; 2#上料OK记忆
LD TR0
AND H50.07  ; 进料2#夹爪NG料
AND W115.11  ; 进料升降伺服取料位
@RSET H56.03  ; 2#上料NG记忆

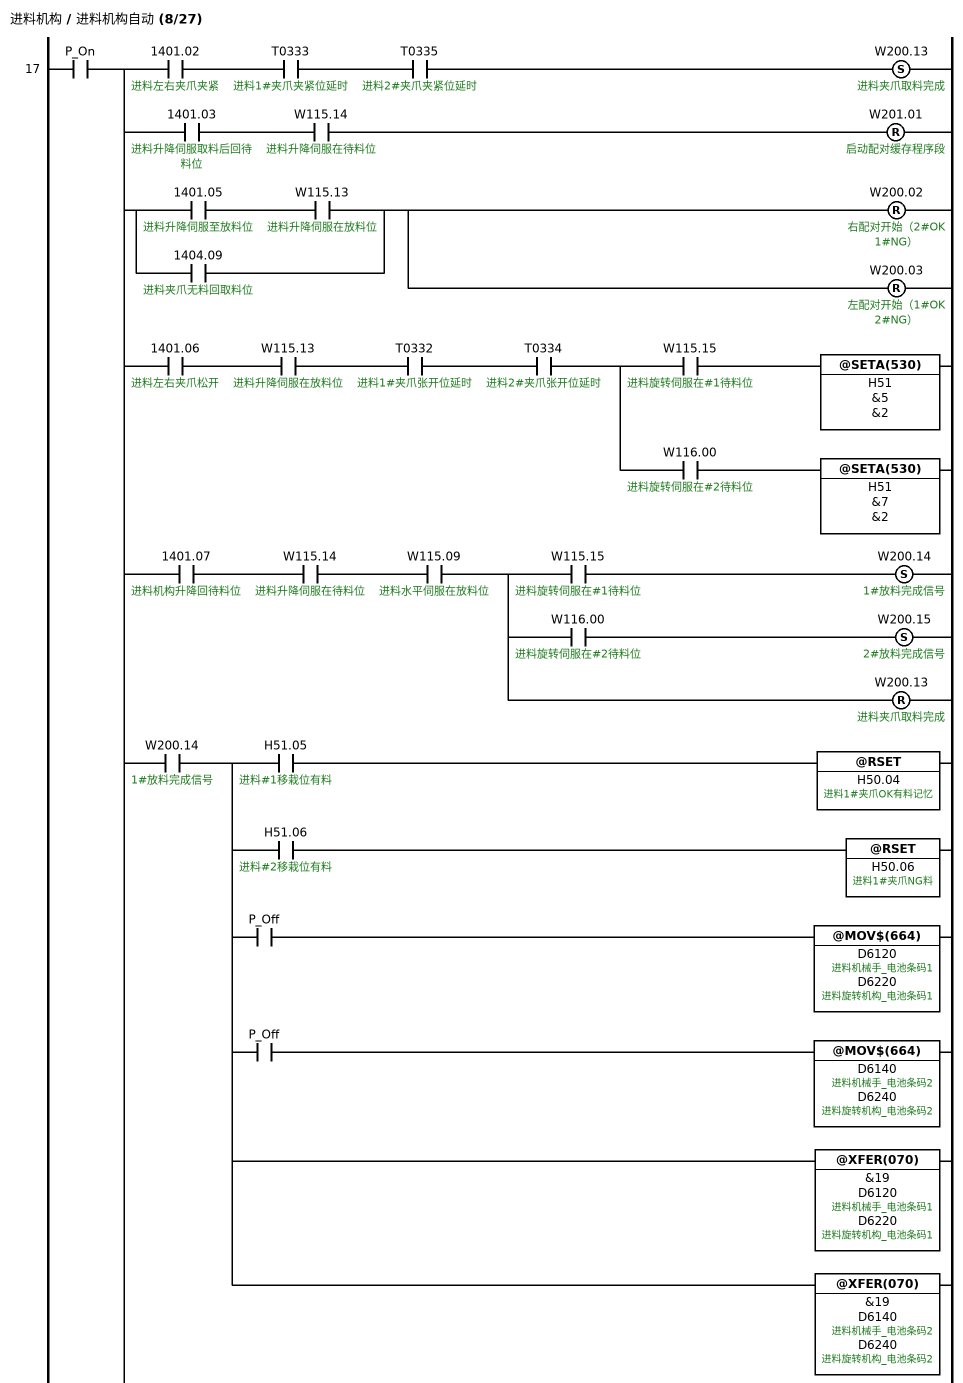

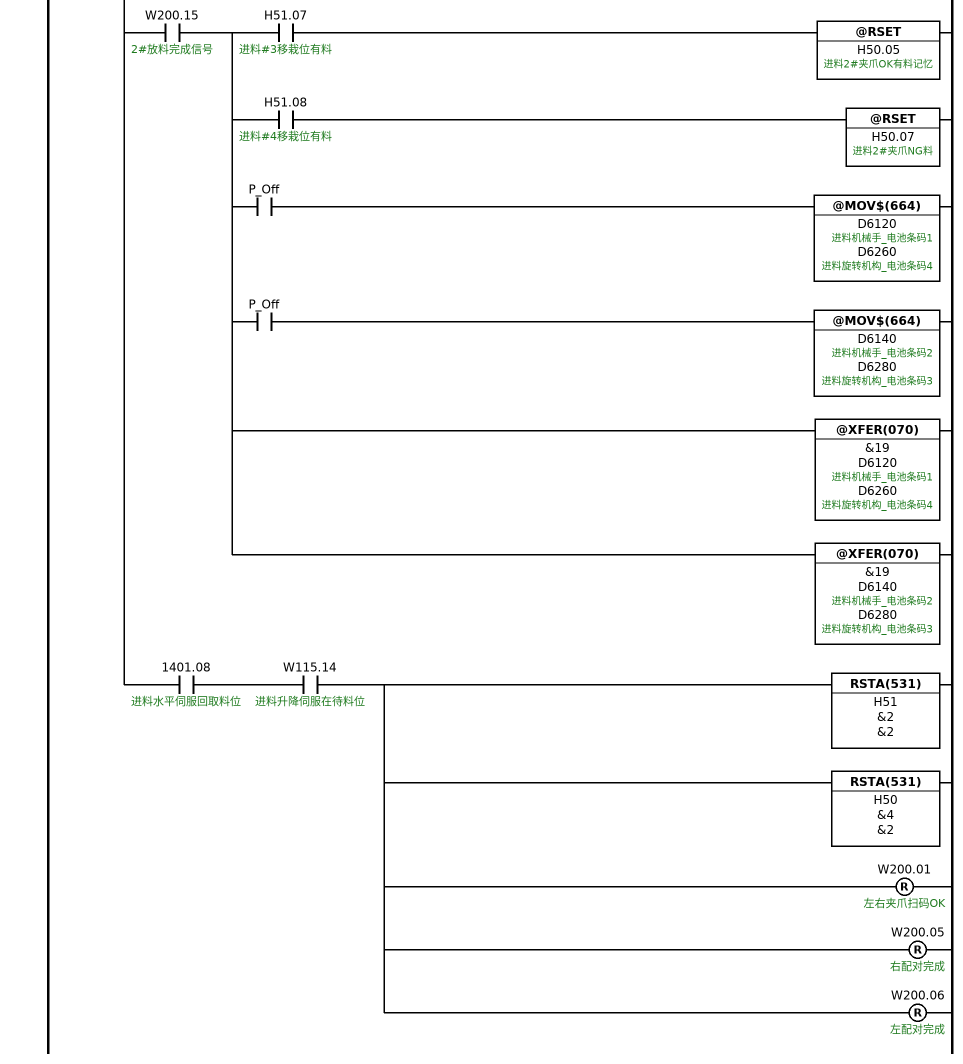
; rung 17
LD P_On
OUT TR0
AND 1401.02  ; 进料左右夹爪夹紧
AND T0333  ; 进料1#夹爪夹紧位延时
AND T0335  ; 进料2#夹爪夹紧位延时
SET W200.13  ; 进料夹爪取料完成
LD TR0
AND 1401.03  ; 进料升降伺服取料后回待料位
AND W115.14  ; 进料升降伺服在待料位
RSET W201.01  ; 启动配对缓存程序段
LD TR0
LD 1401.05  ; 进料升降伺服至放料位
AND W115.13  ; 进料升降伺服在放料位
OR 1404.09  ; 进料夹爪无料回取料位
ANDLD
RSET W200.02  ; 右配对开始（2#OK 1#NG）
RSET W200.03  ; 左配对开始（1#OK 2#NG）
LD TR0
AND 1401.06  ; 进料左右夹爪松开
AND W115.13  ; 进料升降伺服在放料位
AND T0332  ; 进料1#夹爪张开位延时
AND T0334  ; 进料2#夹爪张开位延时
OUT TR1
AND W115.15  ; 进料旋转伺服在#1待料位
@SETA(530) H51 &5 &2
LD TR1
AND W116.00  ; 进料旋转伺服在#2待料位
@SETA(530) H51 &7 &2
LD TR0
AND 1401.07  ; 进料机构升降回待料位
AND W115.14  ; 进料升降伺服在待料位
AND W115.09  ; 进料水平伺服在放料位
OUT TR1
AND W115.15  ; 进料旋转伺服在#1待料位
SET W200.14  ; 1#放料完成信号
LD TR1
AND W116.00  ; 进料旋转伺服在#2待料位
SET W200.15  ; 2#放料完成信号
LD TR1
RSET W200.13  ; 进料夹爪取料完成
LD TR0
AND W200.14  ; 1#放料完成信号
OUT TR1
AND H51.05  ; 进料#1移栽位有料
@RSET H50.04  ; 进料1#夹爪OK有料记忆
LD TR1
AND H51.06  ; 进料#2移栽位有料
@RSET H50.06  ; 进料1#夹爪NG料
LD TR1
AND P_Off
@MOV$(664) D6120 D6220  ; 进料机械手_电池条码1, 进料旋转机构_电池条码1
LD TR1
AND P_Off
@MOV$(664) D6140 D6240  ; 进料机械手_电池条码2, 进料旋转机构_电池条码2
LD TR1
@XFER(070) &19 D6120 D6220  ; 进料机械手_电池条码1, 进料旋转机构_电池条码1
@XFER(070) &19 D6140 D6240  ; 进料机械手_电池条码2, 进料旋转机构_电池条码2
LD TR0
AND W200.15  ; 2#放料完成信号
OUT TR1
AND H51.07  ; 进料#3移栽位有料
@RSET H50.05  ; 进料2#夹爪OK有料记忆
LD TR1
AND H51.08  ; 进料#4移栽位有料
@RSET H50.07  ; 进料2#夹爪NG料
LD TR1
AND P_Off
@MOV$(664) D6120 D6260  ; 进料机械手_电池条码1, 进料旋转机构_电池条码4
LD TR1
AND P_Off
@MOV$(664) D6140 D6280  ; 进料机械手_电池条码2, 进料旋转机构_电池条码3
LD TR1
@XFER(070) &19 D6120 D6260  ; 进料机械手_电池条码1, 进料旋转机构_电池条码4
@XFER(070) &19 D6140 D6280  ; 进料机械手_电池条码2, 进料旋转机构_电池条码3
LD TR0
AND 1401.08  ; 进料水平伺服回取料位
AND W115.14  ; 进料升降伺服在待料位
RSTA(531) H51 &2 &2
RSTA(531) H50 &4 &2
RSET W200.01  ; 左右夹爪扫码OK
RSET W200.05  ; 右配对完成
RSET W200.06  ; 左配对完成

